Universal Robots PolyScope program: Floor Corner Extended.urp

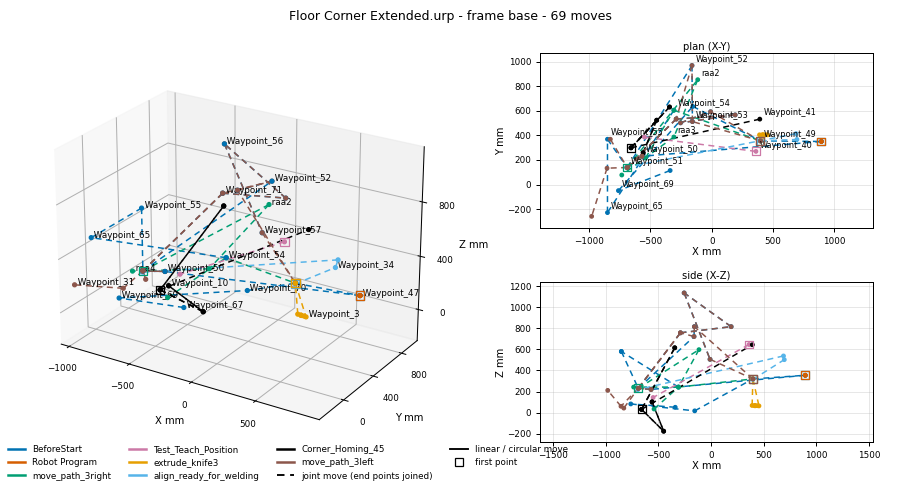
[picture p0: tool path of Floor Corner Extended.urp in frame base, 69 of 124 moves have a stored position in this frame; points joined in program order, loops and branches not executed]
Program Floor Corner Extended (installation=default directory=/programs/UPF createdIn=5.14.5 lastSavedIn=5.14.5 robotSerialNumber=20236801216)
Calibrated DH parameters: a=[-0.000021, -0.748897, -0.28186, -0.00004, -0.000055, 0]; d=[0.236225, -424.082933, -1564.66872, 1988.95162, 0.159094, 0.153873]; alpha=[1.570844, 0.001002, 0.000337, 1.571488, -1.569996, 0]; deltaTheta=[0, -0.516316, 5.626292, 1.173211, 0.000001, 0]
InitVariablesNode variables(variable(name=freedrive_m_var, expression=False))
BeforeStart
  Folder Safe Home Folder
    'if robot is not at home, send it back to home safely'
    'make sure the tcp is welder'
    Set NoAction tcp=pretend_welder
    sp := get_actual_tcp_pose()
    MoveL speed 250 mm/s, acceleration 1200 mm/s^2 (useActiveTCP=true) feature=Base
      Waypoint Variable (Variable): variable=sp
      'if first move is to a variable, skip automove'
    'turn off welder'
    URCap WireTank Serial (WireTank Serial, WireTank, LLC) dataModel(NODE_TITLE=Serial Bridge uR0, Command=[252,82,48], byte_array=true, OUTPUT_ENTRY=Static, QUERY=false, Variable(key=OUTPUT_VARIABLE, variable(name=HwResp)))
    Set DigitalOutput pin=digital_out[0]; digitalValue=0
    jp := get_actual_joint_positions()
    If sp[0]>0.600
      'if x > 600 then above then home'
      MoveJ speed 60 deg/s, acceleration 80 deg/s^2 (useActiveTCP=true) feature=Base
        Waypoint Waypoint_47: TCP in base x=894.111 y=351.078 z=354.441 mm, rx=2.3264 ry=2.0525 rz=0.0574 rad; joints [-187.182, -67.293, 94.726, 57.522, -0.141, -88.018] deg; TCP offset x=-5.49 y=-328 z=106.39 mm, rx=1.2092 ry=-1.2092 rz=1.2092 rad
      SafeHome (positionOptionType=SPEED_AND_ACCELERATION speed=1.047198 acceleration=1.396263 nextMotionTime=2)
    Else 
      Popup Message (haltProgram=false message=retreating to home inputType=Text)
      'for rules 2-8, finish with oldhome then above then home'
      If -1.74<jp[4] and jp[4]<1.05 and -1.74<jp[3] and jp[3]<1.74
        'if oldhome, test teach, then go straight to oldhome'
      ElseIf sp[0]<-.5 and jp[3]>3.14 and -2.62<jp[4] and jp[4]<-0.87
        'if left side weld approach, left weld approach in reverse'
        MoveJ speed 60 deg/s, acceleration 80 deg/s^2 (useActiveTCP=true) feature=Base
          Waypoint Waypoint_50: TCP in base x=-568.711 y=230.602 z=220.209 mm, rx=-1.5191 ry=-0.5351 rz=0.574 rad; joints [-1.233, -73.308, 139.365, 291.685, -131.758, 87.871] deg
          Waypoint Waypoint_51: TCP in base x=-689.65 y=139.001 z=230.693 mm, rx=-0.852 ry=-1.646 rz=1.646 rad; joints [-65.631, -88.39, 163.033, 285.278, -280.919, 90.062] deg
          Waypoint Waypoint_52: TCP in base x=-160.992 y=970.528 z=722.037 mm, rx=-0.555 ry=0.1065 rz=0.3285 rad; joints [-74.362, -75.728, 129.393, 212.138, -169.184, 55.164] deg
          Waypoint Waypoint_53: TCP in base x=-157.624 y=513.351 z=815.67 mm, rx=-0.6727 ry=-1.8523 rz=-0.0554 rad; joints [-158.576, -104.315, 132.512, 57.998, -61.68, -46.426] deg
      ElseIf sp[0]<0 and 0<jp[3] and jp[3]<1.74 and 0.87<jp[4] and jp[4]<2.62
        'if right side around, move back then wapoint 24 then oldhome'
        If sp[0]<-1.0
          xback := p[-1.0,sp[1],sp[2],sp[3],sp[4],sp[5]]
          MoveJ speed 60 deg/s, acceleration 80 deg/s^2 (useActiveTCP=true) feature=Base
            Waypoint Variable (Variable): variable=xback
        MoveJ speed 60 deg/s, acceleration 80 deg/s^2 (useActiveTCP=true) feature=Base
          Waypoint Waypoint_54: TCP in base x=-308.528 y=606.081 z=242.371 mm, rx=-2.1337 ry=0.3494 rz=2.131 rad; joints [-112.4, -74.451, 126.505, 42.726, 91.418, 81.282] deg
      ElseIf jp[3]>2.62 and jp[4]<-3.84
        'if left side second half, then left weld ending sequence'
        If jp[5]<0.35
          MoveJ speed 60 deg/s, acceleration 80 deg/s^2 (useActiveTCP=true) feature=Base
            Waypoint Waypoint_65: TCP in base x=-850.3 y=-229.061 z=580.194 mm, rx=-0.0667 ry=-1.5664 rz=-0.0455 rad; joints [6.605, -69.14, 152.414, 186.359, -269.256, -10.612] deg
        MoveJ speed 60 deg/s, acceleration 80 deg/s^2 (useActiveTCP=true) feature=Base
          SuppressedNode
            Waypoint Waypoint_61: TCP in base x=-1224.453 y=315.135 z=45.036 mm, rx=0.4556 ry=-1.5209 rz=0.4778 rad; joints [-38.105, -18.537, 102.715, 186.465, -269.531, 72.317] deg
          SuppressedNode
            Waypoint Waypoint_62: TCP in base x=-1246.058 y=121.907 z=25.888 mm, rx=-0.7807 ry=-1.4195 rz=-0.7637 rad; joints [-2.239, -16.844, 100.196, 185.863, -269.635, -54.527] deg
          SuppressedNode
            Waypoint Waypoint_63: TCP in base x=-850.3 y=142.696 z=580.194 mm, rx=-0.0667 ry=-1.5664 rz=-0.0455 rad; joints [-33.715, -70.118, 156.539, 183.763, -269.222, 29.711] deg
          SuppressedNode
            Waypoint Waypoint_64: TCP in base x=-850.307 y=-229.065 z=580.197 mm, rx=-0.0667 ry=-1.5664 rz=-0.0455 rad; joints [6.605, -69.141, 152.414, 186.36, -269.255, -10.612] deg
          'above is testing, below is real'
          Waypoint Waypoint_55: TCP in base x=-850.296 y=369.354 z=580.191 mm, rx=-0.0667 ry=-1.5664 rz=-0.0455 rad; joints [-51.358, -68.674, 149.321, 189.759, -269.326, 47.358] deg
          SuppressedNode
            Waypoint Waypoint_60: TCP in base x=-826.865 y=369.366 z=43.112 mm, rx=0.575 ry=-1.4922 rz=0.5971 rad; joints [-59.177, -17.074, 121.534, 166.294, -269.929, 102.173] deg
          Waypoint Waypoint_59: motionParameters(nextMotionTime=2); TCP in base x=-689.651 y=138.973 z=230.7 mm, rx=-0.852 ry=-1.646 rz=1.646 rad; joints [-65.63, -88.392, 163.034, 285.278, -280.919, 90.062] deg
          Waypoint Waypoint_71: TCP in base x=-289.685 y=534.258 z=757.199 mm, rx=-0.2952 ry=-0.653 rz=0.3894 rad; joints [-79.881, -94.829, 156.624, 238.16, -217.621, 99.184] deg
          Waypoint Waypoint_58: TCP in base x=191.12 y=567.518 z=815.513 mm, rx=-0.1358 ry=0.3961 rz=0.2088 rad; joints [-94.611, -101.484, 149.999, 189.458, -152.19, 49.064] deg
          Waypoint Waypoint_56: TCP in base x=-254.568 y=502.959 z=1135.401 mm, rx=-0.2619 ry=-0.7497 rz=1.3491 rad; joints [-116.567, -108.934, 141.5, 126.12, -66.905, -29.189] deg
          Waypoint Waypoint_57: TCP in base x=-9.221 y=593.713 z=505.809 mm, rx=-1.4244 ry=-2.3441 rz=-0.5276 rad; joints [-167.352, -114.202, 136.688, 39.052, -32.592, -65.93] deg
      ElseIf jp[3]<-2.09
        'bottom homing'
        MoveJ speed 60 deg/s, acceleration 80 deg/s^2 (useActiveTCP=true) feature=Base
          SuppressedNode
            Waypoint Waypoint_66: TCP in base x=-1189.333 y=-102.843 z=-176.058 mm, rx=1.1963 ry=-1.1853 rz=1.2301 rad; joints [-19.887, -1.876, 78.341, -165.92, 91.498, 110.543] deg
          ''
          If sp[0]<-0.95
            xback := p[-0.95,sp[1],sp[2],sp[3],sp[4],sp[5]]
            MoveL speed 250 mm/s, acceleration 1200 mm/s^2 (useActiveTCP=true) feature=Base
              Waypoint Variable (Variable): variable=xback
          Waypoint Waypoint_67: TCP in base x=-339.169 y=114.271 z=51.007 mm, rx=-0.4342 ry=1.8727 rz=-1.8852 rad; joints [-80.817, -56.025, 141.954, -98.756, -22.671, 103.625] deg
      ElseIf jp[3]<0 and jp[4]<-3.14
        'if left side homing, special unspin'
        MoveJ speed 60 deg/s, acceleration 80 deg/s^2 (useActiveTCP=true) feature=Base
          SuppressedNode
            Waypoint Waypoint_68: TCP in base x=-1436.144 y=-207.487 z=20.65 mm, rx=-1.0168 ry=-1.7024 rz=1.6295 rad; joints [2.271, -43.137, 96.498, -42.2, -211.884, 93.908] deg
          ''
          Waypoint Waypoint_69: TCP in base x=-760.827 y=-49.763 z=82.65 mm, rx=-1.0262 ry=-1.6127 rz=1.5471 rad; joints [-12.694, -64.084, 157.914, -89.201, -220.703, 89.352] deg
          Waypoint Waypoint_70: TCP in base x=-154.415 y=636.923 z=16.979 mm, rx=-0.3028 ry=1.487 rz=0.1222 rad; joints [-64.641, -61.184, 139.176, -160.395, -91.873, 99.702] deg
      ElseIf (sp[4]<-3 or sp[4]>3) and -0.02<sp[5] and sp[5]<0.02
        'go straight to home'
      ElseIf 2>1
        'if none of the other options, then error continuously'
        Loop While (checkContinuously=false) expression=2>1
          Popup Message (haltProgram=false message=Unknown Position. Find Calvin for Assistance inputType=Text)
      'insert logic for how to get back to oldhome'
      'finish with oldhome then above then home'
      MoveJ speed 60 deg/s, acceleration 80 deg/s^2 (useActiveTCP=true) feature=Base
        Waypoint Waypoint_49: motionParameters(jointSpeed=1.047198 jointAcceleration=1.396263 cartesianSpeed=0.25 cartesianAcceleration=1.2); TCP in base x=397.354 y=356.263 z=319.809 mm, rx=2.3163 ry=2.0576 rz=0.0741 rad; joints [-198.126, -117.851, 133.304, -13.008, -11.424, -6.036] deg
        Waypoint Waypoint_48: TCP in base x=894.09 y=351.09 z=354.453 mm, rx=2.3264 ry=2.0525 rz=0.0573 rad; joints [-187.181, -67.294, 94.727, 57.523, -0.141, -88.018] deg
      SafeHome (positionOptionType=SPEED_AND_ACCELERATION speed=1.047198 acceleration=1.396263 nextMotionTime=2)
Robot Program (runOnlyOnce=true)
  'start of main program'
  Set NoAction tcp=pretend_welder
  SafeHome (positionOptionType=SPEED_AND_ACCELERATION speed=1.047198 acceleration=1.396263 nextMotionTime=2)
  Script file /programs/analyze_touchpoints.script
    | # this file creates the function for analyzing touchpoints
    | # define pi
    | pi = 3.1415926535
    | 
    | # this is the main entry point for calculations.
    | # it takes in the 5 points, analyzes the shape of the box, and then calculates path points and returns them
    | # specifically for Down, Over, then Around (DOtA)
    | # specifically for right-sided boxes (vertical weld on right side of edge)
    | def main_calculate_right(p11, p12, p21, p22, p3, p13, p23, chamferover):
    |     struct1 = analyze_touchpoints_only(p11, p12, p21, p22, p3)
    |     list1 = analyze_vertical_touchpoints(p11, p12, p13, p21, p22, p23, p3)
    |     struct2 = calculate_DOtA_points_right(struct1, list1, chamferover)
    |     validity = check_validity_right(struct1, struct2)
    |     return struct2
    | end
    | 
    | # this is the main entry point for calculations.
    | # it takes in the 5 points, analyzes the shape of the box, and then calculates path points and returns them
    | # specifically for Down, Over, then Around (DOtA)
    | # specifically for left-sided boxes (vertical weld on left side of edge)
    | def main_calculate_left(p11, p12, p21, p22, p3, p13, p23, chamferover):
    |     struct1 = analyze_touchpoints_only(p11, p12, p21, p22, p3)
    |     list1 = analyze_vertical_touchpoints(p11, p12, p13, p21, p22, p23, p3)
    |     struct2 = calculate_DOtA_points_left(struct1, list1, chamferover)
    |     validity = check_validity_left(struct1, struct2)
    |     return struct2
    | end
    | 
    | # this is the main entry point for calculations, for Floor Corner Extended.
    | # it takes in the 7 touchpoints, analyzes the shape of the box.
    | # takes in the user defined point for the top of the weld (tcp_pose_top) and then calculates path points
    | # loopingly tries to calculate the extension along the sidewall that fulfills get_inverse_kin_has_solution() and provides the farthest extension possible
    | # returns the pathpoints
    | # specifically for Down, Over, then Around (DOtA)
    | # specifically for right-sided boxes (vertical weld on right side of edge)
    | def main_calculate_right_extended(p11, p12, p21, p22, p3, p13, p23, chamferover, tcp_pose_top):
    |     struct1 = analyze_touchpoints_only(p11, p12, p21, p22, p3)
    |     list1 = analyze_vertical_touchpoints(p11, p12, p13, p21, p22, p23, p3)
    |     struct2 = calculate_DOtA_points_right_extended(struct1, list1, chamferover, tcp_pose_top)
    |     validity = check_validity_right(struct1, struct2)
    |     return struct2
    | end
    | 
    | # this is the main entry point for calculations, for Floor Corner Extended.
    | # it takes in the 7 touchpoints, analyzes the shape of the box.
    | # takes in the user defined point for the top of the weld (tcp_pose_top) and then calculates path points
    | # loopingly tries to calculate the extension along the sidewall that fulfills get_inverse_kin_has_solution() and provides the farthest extension possible
    | # returns the pathpoints
    | # specifically for Down, Over, then Around (DOtA)
    | # specifically for left-sided boxes (vertical weld on left side of edge)
    | def main_calculate_left_extended(p11, p12, p21, p22, p3, p13, p23, chamferover, tcp_pose_top):
    |     struct1 = analyze_touchpoints_only(p11, p12, p21, p22, p3)
    |     list1 = analyze_vertical_touchpoints(p11, p12, p13, p21, p22, p23, p3)
    |     struct2 = calculate_DOtA_points_left_extended(struct1, list1, chamferover, tcp_pose_top)
    |     validity = check_validity_left(struct1, struct2)
    |     return struct2
    | end
    | 
    | # it takes 5 arguments as points
    | # it returns a struct containing: (pointintersect, pointapproach1, pointapproach2, point1, point2, point3, point4, point5, pointreturn1, heading1, heading2, heading3, path2r1, path2r2, path2l1, path2l2)
    | # specifically for Around then Up (AtU)
    | def analyze_touchpoints(p11, p12, p21, p22, p3):
    |   # FIND THE INTERSECTION
    |   # comment get the z
    |   zcoord=p3[2]
    | 
    |   # get the raw points from the first line
    |   l1p1x=p11[0]
    |   l1p1y=p11[1]
    |   l1p2x=p12[0]
    |   l1p2y=p12[1]
    | 
    |   # equate the first line in 2d space
    |   ml1 = (l1p2y-l1p1y) / (l1p2x-l1p1x)
    | 
    |   # b = y - mx
    |   bl1 = l1p1y - ml1 * l1p1x
    | 
    |   # get the raw points from the second line
    |   l2p1x=p21[0]
    |   l2p1y=p21[1]
    |   l2p2x=p22[0]
    |   l2p2y=p22[1]
    | 
    |   # equate the second line in 2d space
    |   ml2 = (l2p2y-l2p1y) / (l2p2x-l2p1x)
    | 
    |   # b = y - mx
    |   bl2 = l2p1y - ml2 * l2p1x
    | 
    | 
    |   # find the intersection of the two lines
    |   # m1x+b1 = m2x+b2
    |   # m1x - m2x = b2 - b1
    |   # x = (b2-b1) / (m1-m2)
    |   xintersect = (bl2-bl1) / (ml1-ml2)
    |   yintersect = ml1 * xintersect + bl1
    | 
    |   #FIND THE VECTORS
    |   #define a vector from the intersection to the second point on the first line
    |   l1delxfull = l1p2x - xintersect
    |   l1delyfull = l1p2y - yintersect
    | 
    |   l1delmag = sqrt(l1delxfull*l1delxfull + l1delyfull*l1delyfull)
    | 
    |   l1delxunit = l1delxfull / l1delmag
    |   l1delyunit = l1delyfull / l1delmag
    | 
    |   #define a vector from the intersection to the second point on the second line
    |   l2delxfull = l2p2x - xintersect
    |   l2delyfull = l2p2y - yintersect
    | 
    |   l2delmag = sqrt(l2delxfull*l2delxfull + l2delyfull*l2delyfull)
    | 
    |   l2delxunit = l2delxfull / l2delmag
    |   l2delyunit = l2delyfull / l2delmag
    | 
    |   # FIND THE FOUR POINTS ON THE LINES
    |   # find locations 8 inches away from  intersect point
    |   # CONST
    |   welddistance = 8
    |   roundoverdistance = 0.05
    |   zup = .375
    |   # inches
    |   wd = welddistance * 25.4 / 1000
    |   rod = roundoverdistance * 25.4 / 1000
    |   zup = zup * 25.4 / 1000
    | 
    |   # now we have the unit vector. extend the weld distance from the intersection
    |   x = xintersect + l1delxunit * wd
    |   y = yintersect + l1delyunit * wd
    |   z = zcoord + zup
    | 
    |   point1 = p[x,y,z,1.570796,0,0] # dummy orientation for now
    | 
    |   x = xintersect + l1delxunit * rod
    |   y = yintersect + l1delyunit * rod
    | 
    |   point2 = p[x,y,z,1.570796,0,0]
    | 
    |   # now we have the unit vector. extend the weld distance from the intersection
    |   x = xintersect + l2delxunit * wd
    |   y = yintersect + l2delyunit * wd
    | 
    |   point5 = p[x,y,z,0,-1.570796,0]
    | 
    |   x = xintersect + l2delxunit * rod
    |   y = yintersect + l2delyunit * rod
    | 
    |   point4 = p[x,y,z,0,-1.570796,0]
    | 
    |   #DEFINE APPROACH POINTS
    |   pointintersect = p[xintersect,yintersect,zcoord,0,0,0]
    |   pointapproach1 = p[xintersect+0.1,yintersect+0.1,z,1.570796,0,0]
    |   pointapproach2 = p[point1[0], point1[1]+0.1, point1[2], point1[3], point1[4], point1[5]]
    |   pointreturn1 = p[point5[0]+0.1, point5[1], point5[2], point5[3], point5[4], point5[5]]
    | 
    |   #FIND HEADINGS
    |   #for each heading, find the angle of the line with respect to the pos x axis. then add/subtract 90 degrees because you want to be perpendicular to that
    |   headingvector1 = convert_uv_to_heading(l1delxunit, l1delyunit)
    |   headingvector2 = convert_uv_to_heading(l2delxunit, l2delyunit)
    |   # find halfway heading
    |   heading2 = (headingvector1 + headingvector2)/2
    |   # find headings that the robot should face while traveling, perpendicular to the vectors of the sides of the box
    |   heading1 = headingvector1 + pi/2
    |   heading3 = headingvector2 - pi/2
    | 
    |   #FIND POINT 3
    |   #see if we have to / can find point 3
    |   findpoint3 = True
    |   if roundoverdistance == 0:
    |     findpoint3 = False
    |   end
    |   if findpoint3:
    |     # i need to find the point3 such that the arc from p2 to p3 to p4 is tangent to p1-p2 and p4-p5. making this a smooth path will be good
    |     # the direction of movement is from pointintersect in the direction of heading2
    |     # how much movement though? this will depend on whether it is actually a 90 degree angle or not.
    |     # first, find the perpendicular lines through points 2 and 4
    |     perp2 = find_perpendicular_line(ml1, point2[0], point2[1])
    |     perp4 = find_perpendicular_line(ml2, point4[0], point4[1])
    |     # next, find the intersection of those two lines
    |     perpintersect = find_intersection(perp2[0], perp2[1], perp4[0], perp4[1])
    |     radiusofcircle = distance_between(perpintersect[0], perpintersect[1], 0, point2[0], point2[1], 0)
    |     # find a vector the direction of heading2
    |     uvx = cos(heading2)
    |     uvy = sin(heading2)
    |     # compute point3. pass in negative radius because the direction is into the tank but we want to move from the intersection out to the rounded edge
    |     point3coords = add_vectordistance_to_point(perpintersect[0], perpintersect[1], z, uvx, uvy, 0, -1 * radiusofcircle)
    |     point3 = p[point3coords[0], point3coords[1], point3coords[2], 0, 0, 0]
    |   end
    | 
    |   #APPLY ACTUAL RXRYRZ TO POINTS
    |   # convert the headings to rxryrz and insert those values into the relevant points
    |   rxryrz = convert_heading_to_axang(heading1)
    |   rx = rxryrz[0]
    |   ry = rxryrz[1]
    |   rz = rxryrz[2]
    |   pointapproach1 = p[pointapproach1[0], pointapproach1[1], pointapproach1[2], rx, ry, rz]
    |   pointapproach2 = p[pointapproach2[0], pointapproach2[1], pointapproach2[2], rx, ry, rz]
    |   point1 = p[point1[0], point1[1], point1[2], rx, ry, rz]
    |   point2 = p[point2[0], point2[1], point2[2], rx, ry, rz]
    |   rxryrz = convert_heading_to_axang(heading2)
    |   rx = rxryrz[0]
    |   ry = rxryrz[1]
    |   rz = rxryrz[2]
    |   if findpoint3:
    |     point3 = p[point3[0], point3[1], point3[2], rx, ry, rz]
    |   else:
    |     point3 = point2
    |   end
    |   rxryrz = convert_heading_to_axang(heading3)
    |   rx = rxryrz[0]
    |   ry = rxryrz[1]
    |   rz = rxryrz[2]
    |   point4 = p[point4[0], point4[1], point4[2], rx, ry, rz]
    |   point5 = p[point5[0], point5[1], point5[2], rx, ry, rz]
    |   pointreturn1 = p[pointreturn1[0], pointreturn1[1], pointreturn1[2], rx, ry, rz]
    | 
    |   #find path2 (the part that goes up)
    |   four_vertical_points = find_vertical_points(pointintersect, l1delxunit, l1delyunit, l2delxunit, l2delyunit, zup, wd, heading1, heading3)
    |   path2r1 = four_vertical_points[0]
    |   path2r2 = four_vertical_points[1]
    |   path2l1 = four_vertical_points[2]
    |   path2l2 = four_vertical_points[3]
    | 
    |   #RETURN STRUCT
    |   ret = struct(pointintersect=pointintersect, pointapproach1=pointapproach1, pointapproach2=pointapproach2, point1=point1, point2=point2, point3=point3, point4=point4, point5=point5, pointreturn1=pointreturn1, heading1=heading1, heading2=heading2, heading3=heading3, path2r1=path2r1, path2r2=path2r2, path2l1=path2l1, path2l2=path2l2)
    |   return ret
    | end
    | 
    | # it takes 5 arguments as points
    | # it returns a struct containing: (pointintersect, heading1, heading2, heading3, l1delxunit, l1delyunit, l2delxunit, l2delyunit)
    | def analyze_touchpoints_only(p11, p12, p21, p22, p3):
    |   # FIND THE INTERSECTION
    |   # comment get the z
    |   zcoord=p3[2]
    | 
    |   # get the raw points from the first line
    |   l1p1x=p11[0]
    |   l1p1y=p11[1]
    |   l1p2x=p12[0]
    |   l1p2y=p12[1]
    | 
    |   # equate the first line in 2d space
    |   ml1 = (l1p2y-l1p1y) / (l1p2x-l1p1x)
    | 
    |   # b = y - mx
    |   bl1 = l1p1y - ml1 * l1p1x
    | 
    |   # get the raw points from the second line
    |   l2p1x=p21[0]
    |   l2p1y=p21[1]
    |   l2p2x=p22[0]
    |   l2p2y=p22[1]
    | 
    |   # equate the second line in 2d space
    |   ml2 = (l2p2y-l2p1y) / (l2p2x-l2p1x)
    | 
    |   # b = y - mx
    |   bl2 = l2p1y - ml2 * l2p1x
    | 
    | 
    |   # find the intersection of the two lines
    |   # m1x+b1 = m2x+b2
    |   # m1x - m2x = b2 - b1
    |   # x = (b2-b1) / (m1-m2)
    |   xintersect = (bl2-bl1) / (ml1-ml2)
    |   yintersect = ml1 * xintersect + bl1
    | 
    |   pointintersect = p[xintersect,yintersect,zcoord,0,0,0]
    | 
    |   #FIND THE VECTORS
    |   #define a vector from the intersection to the second point on the first line
    |   l1delxfull = l1p2x - xintersect
    |   l1delyfull = l1p2y - yintersect
    | 
    |   l1delmag = sqrt(l1delxfull*l1delxfull + l1delyfull*l1delyfull)
    | 
    |   l1delxunit = l1delxfull / l1delmag
    |   l1delyunit = l1delyfull / l1delmag
    | 
    |   #define a vector from the intersection to the second point on the second line
    |   l2delxfull = l2p2x - xintersect
    |   l2delyfull = l2p2y - yintersect
    | 
    |   l2delmag = sqrt(l2delxfull*l2delxfull + l2delyfull*l2delyfull)
    | 
    |   l2delxunit = l2delxfull / l2delmag
    |   l2delyunit = l2delyfull / l2delmag
    | 
    |   #FIND HEADINGS
    |   #for each heading, find the angle of the line with respect to the pos x axis. then add/subtract 90 degrees because you want to be perpendicular to that
    |   headingvector1 = convert_uv_to_heading(l1delxunit, l1delyunit)
    |   headingvector2 = convert_uv_to_heading(l2delxunit, l2delyunit)
    |   # find halfway heading
    |   heading2 = (headingvector1 + headingvector2)/2
    |   # find headings that the robot should face while traveling, perpendicular to the vectors of the sides of the box
    |   heading1 = headingvector1 + pi/2
    |   heading3 = headingvector2 - pi/2
    | 
    |   #RETURN STRUCT
    |   ret = struct(pointintersect=pointintersect, heading1=heading1, heading2=heading2, heading3=heading3, l1delxunit=l1delxunit, l1delyunit=l1delyunit, l2delxunit=l2delxunit, l2delyunit=l2delyunit)
    |   return ret
    | end
    | 
    | # given a struct from analyze_touchpoints_only(), calculate the points
    | # for right, for non-extended
    | def calculate_DOtA_points_right(struct1, listleans, chamferover):
    |     # get the stuff from the struct
    |     pointintersect = struct1[0]
    |     heading1 = struct1[1]
    |     heading2 = struct1[2]
    |     heading3 = struct1[3]
    |     l1delxunit = struct1[4]
    |     l1delyunit = struct1[5]
    |     l2delxunit = struct1[6]
    |     l2delyunit = struct1[7]
    | 
    |     # FIND THE POINTS ON THE LINES OF THE FIRST TURN PATH
    |     # find locations 8 inches away from  intersect point
    |     # CONST
    |     welddistance1 = 8 # vertical weld distance
    |     welddistance2 = 6 # first path second leg
    |     welddistance3 = 8 # second path second leg
    |     zup = .375
    |     # inches
    |     wd1 = welddistance1 * 25.4 / 1000
    |     wd2 = welddistance2 * 25.4 / 1000
    |     wd3 = welddistance3 * 25.4 / 1000
    |     zup = zup * 25.4 / 1000
    |     chamferovermm =  chamferover * 25.4 / 1000
    | 
    |     x = pointintersect[0] + l1delxunit * chamferovermm
    |     y = pointintersect[1] + l1delyunit * chamferovermm
    |     z = pointintersect[2] + zup
    | 
    |     #apply actual rxryrz to points
    |     # convert the headings to rxryrz and insert those values into the relevant points
    |     rxryrz = convert_heading_to_axang_preheatdown(heading1)
    |     rx = rxryrz[0]
    |     ry = rxryrz[1]
    |     rz = rxryrz[2]
    | 
    |     point1 = p[x + wd1*listleans[0], y + wd1*listleans[1], z + wd1, rx, ry, rz] # add in the listleans factor to follow the face of the box as we move up
    |     point2 = p[x, y, z, rx, ry, rz]
    | 
    |     # convert the headings to rxryrz and insert those values into the relevant points
    |     rxryrz = convert_heading_to_axang_ccw(heading1)
    |     rx = rxryrz[0]
    |     ry = rxryrz[1]
    |     rz = rxryrz[2]
    | 
    |     point4 = p[x, y, z, rx, ry, rz]
    |     x = x + l1delxunit * wd2
    |     y = y + l1delyunit * wd2
    |     point5 = p[x, y, z, rx, ry, rz]
    | 
    |     # FIND THE POINTS ON THE LINES OF THE SECOND AROUND PATH
    |     roundoverdistance = 0.05
    |     rod = roundoverdistance * 25.4 / 1000
    | 
    |     # now we have the unit vector. extend the weld distance from the intersection
    |     x = pointintersect[0] + l1delxunit * chamferovermm
    |     y = pointintersect[1] + l1delyunit * chamferovermm
    |     # convert the headings to rxryrz and insert those values into the relevant points
    |     rxryrz = convert_heading_to_axang(heading1)
    |     rx = rxryrz[0]
    |     ry = rxryrz[1]
    |     rz = rxryrz[2]
    |     point_1 = p[x, y, z, rx, ry, rz]
    | 
    |     x = pointintersect[0] + l1delxunit * rod
    |     y = pointintersect[1] + l1delyunit * rod
    |     point_2 = p[x, y, z, rx, ry, rz]
    | 
    |     # now we have the unit vector. extend the weld distance from the intersection
    |     x = pointintersect[0] + l2delxunit * wd3
    |     y = pointintersect[1] + l2delyunit * wd3
    |     # convert the headings to rxryrz and insert those values into the relevant points
    |     rxryrz = convert_heading_to_axang(heading3)
    |     rx = rxryrz[0]
    |     ry = rxryrz[1]
    |     rz = rxryrz[2]
    |     point_5 = p[x, y, z, rx, ry, rz]
    | 
    |     x = pointintersect[0] + l2delxunit * rod
    |     y = pointintersect[1] + l2delyunit * rod
    |     point_4 = p[x, y, z, rx, ry, rz]
    | 
    |     #FIND POINT 3
    |     # by calling analyze_touchpoints()
    |     atret = analyze_touchpoints(point_2, point_1, point_4, point_5, pointintersect)
    |     point_3 = atret[5]
    | 
    | 
    |     struct2 = struct(point1=point1, point2=point2, point4=point4, point5=point5, point_1=point_1, point_2=point_2, point_3=point_3, point_4=point_4, point_5=point_5)
    |     return struct2
    | end
    | 
    | # given a struct from analyze_touchpoints_only(), calculate the points
    | # for left, for non-extended
    | def calculate_DOtA_points_left(struct1, listleans, chamferover):
    |     # get the stuff from the struct
    |     pointintersect = struct1[0]
    |     heading1 = struct1[1]
    |     heading2 = struct1[2]
    |     heading3 = struct1[3]
    |     l1delxunit = struct1[4]
    |     l1delyunit = struct1[5]
    |     l2delxunit = struct1[6]
    |     l2delyunit = struct1[7]
    | 
    |     # FIND THE POINTS ON THE LINES OF THE FIRST TURN PATH
    |     # find locations 8 inches away from  intersect point
    |     # CONST
    |     welddistance1 = 8 # vertical weld distance
    |     welddistance2 = 6 # first path second leg
    |     welddistance3 = 8 # second path second leg
    |     zup = .375
    |     # inches
    |     wd1 = welddistance1 * 25.4 / 1000
    |     wd2 = welddistance2 * 25.4 / 1000
    |     wd3 = welddistance3 * 25.4 / 1000
    |     zup = zup * 25.4 / 1000
    |     chamferovermm =  chamferover * 25.4 / 1000
    | 
    |     x = pointintersect[0] + l2delxunit * chamferovermm
    |     y = pointintersect[1] + l2delyunit * chamferovermm
    |     z = pointintersect[2] + zup
    | 
    |     #apply actual rxryrz to points
    |     # convert the headings to rxryrz and insert those values into the relevant points
    |     rxryrz = convert_heading_to_axang_preheatdown(heading3)
    |     rx = rxryrz[0]
    |     ry = rxryrz[1]
    |     rz = rxryrz[2]
    | 
    |     point1 = p[x + wd1*listleans[0], y + wd1*listleans[1], z + wd1, rx, ry, rz]
    |     point2 = p[x, y, z, rx, ry, rz]
    | 
    |     # convert the headings to rxryrz and insert those values into the relevant points
    |     rxryrz = convert_heading_to_axang(heading3)
    |     rx = rxryrz[0]
    |     ry = rxryrz[1]
    |     rz = rxryrz[2]
    | 
    |     point4 = p[x, y, z, rx, ry, rz]
    |     x = x + l2delxunit * wd2
    |     y = y + l2delyunit * wd2
    |     point5 = p[x, y, z, rx, ry, rz]
    | 
    |     # FIND THE POINTS ON THE LINES OF THE SECOND AROUND PATH
    |     roundoverdistance = 0.05
    |     rod = roundoverdistance * 25.4 / 1000
    | 
    |     # now we have the unit vector. extend the weld distance from the intersection
    |     x = pointintersect[0] + l2delxunit * chamferovermm
    |     y = pointintersect[1] + l2delyunit * chamferovermm
    |     # convert the headings to rxryrz and insert those values into the relevant points
    |     rxryrz = convert_heading_to_axang_ccw(heading3)
    |     rx = rxryrz[0]
    |     ry = rxryrz[1]
    |     rz = rxryrz[2]
    |     point_1 = p[x, y, z, rx, ry, rz]
    | 
    |     x = pointintersect[0] + l2delxunit * rod
    |     y = pointintersect[1] + l2delyunit * rod
    |     point_2 = p[x, y, z, rx, ry, rz]
    | 
    |     # now we have the unit vector. extend the weld distance from the intersection
    |     x = pointintersect[0] + l1delxunit * wd3
    |     y = pointintersect[1] + l1delyunit * wd3
    |     # convert the headings to rxryrz and insert those values into the relevant points
    |     rxryrz = convert_heading_to_axang_ccw(heading1)
    |     rx = rxryrz[0]
    |     ry = rxryrz[1]
    |     rz = rxryrz[2]
    |     point_5 = p[x, y, z, rx, ry, rz]
    | 
    |     x = pointintersect[0] + l1delxunit * rod
    |     y = pointintersect[1] + l1delyunit * rod
    |     point_4 = p[x, y, z, rx, ry, rz]
    | 
    |     #FIND POINT 3
    |     # by calling analyze_touchpoints()
    |     atret = analyze_touchpoints(point_2, point_1, point_4, point_5, pointintersect)
    |     point_3 = atret[5]
    |     #point 3 will not have the correct rxryrz though because now the gun needs to be face up.
    |     rxryrz = convert_heading_to_axang_ccw(heading2)
    |     rx = rxryrz[0]
    |     ry = rxryrz[1]
    |     rz = rxryrz[2]
    |     point_3 = p[point_3[0], point_3[1], point_3[2], rx, ry, rz]
    | 
    |     struct2 = struct(point1=point1, point2=point2, point4=point4, point5=point5, point_1=point_1, point_2=point_2, point_3=point_3, point_4=point_4, point_5=point_5)
    |     return struct2
    | end
    | 
    | # given a struct from analyze_touchpoints_only(), calculate the points
    | # for right, for extended
    | def calculate_DOtA_points_right_extended(struct1, listleans, chamferover, tcp_pose_top):
    |     # get the stuff from the struct
    |     pointintersect = struct1[0]
    |     heading1 = struct1[1]
    |     heading2 = struct1[2]
    |     heading3 = struct1[3]
    |     l1delxunit = struct1[4]
    |     l1delyunit = struct1[5]
    |     l2delxunit = struct1[6]
    |     l2delyunit = struct1[7]
    | 
    |     # FIND THE POINTS ON THE LINES OF THE FIRST TURN PATH
    |     # find locations 8 inches away from  intersect point
    |     # CONST
    |     # welddistance1 = 8 # vertical weld distance
    |     welddistance2 = 6 # first path second leg
    |     welddistance3 = 8 # second path second leg
    |     zup = .375
    |     # inches
    |     # wd1 = welddistance1 * 25.4 / 1000
    |     wd2 = welddistance2 * 25.4 / 1000
    |     wd3 = welddistance3 * 25.4 / 1000
    |     zup = zup * 25.4 / 1000
    |     chamferovermm =  chamferover * 25.4 / 1000
    | 
    |     # weld distance is the distance that it will weld. this will make it start at the z height that the user specified
    |     wd1 = tcp_pose_top[2] - pointintersect[2] - zup
    | 
    |     x = pointintersect[0] + l1delxunit * chamferovermm
    |     y = pointintersect[1] + l1delyunit * chamferovermm
    |     z = pointintersect[2] + zup
    | 
    |     #apply actual rxryrz to points
    |     # convert the headings to rxryrz and insert those values into the relevant points
    |     rxryrz = convert_heading_to_axang_preheatdown(heading1)
    |     rx = rxryrz[0]
    |     ry = rxryrz[1]
    |     rz = rxryrz[2]
    | 
    |     point1 = p[x + wd1*listleans[0], y + wd1*listleans[1], z + wd1, rx, ry, rz] # add in the listleans factor to follow the face of the box as we move up
    |     point2 = p[x, y, z, rx, ry, rz]
    | 
    |     # convert the headings to rxryrz and insert those values into the relevant points
    |     rxryrz = convert_heading_to_axang_ccw(heading1)
    |     rx = rxryrz[0]
    |     ry = rxryrz[1]
    |     rz = rxryrz[2]
    | 
    |     point4 = p[x, y, z, rx, ry, rz]
    |     x = x + l1delxunit * wd2
    |     y = y + l1delyunit * wd2
    |     point5 = p[x, y, z, rx, ry, rz]
    | 
    |     # FIND THE POINTS ON THE LINES OF THE SECOND AROUND PATH
    |     roundoverdistance = 0.05
    |     rod = roundoverdistance * 25.4 / 1000
    | 
    |     # now we have the unit vector. extend the weld distance from the intersection
    |     x = pointintersect[0] + l1delxunit * chamferovermm
    |     y = pointintersect[1] + l1delyunit * chamferovermm
    |     # convert the headings to rxryrz and insert those values into the relevant points
    |     rxryrz = convert_heading_to_axang(heading1)
    |     rx = rxryrz[0]
    |     ry = rxryrz[1]
    |     rz = rxryrz[2]
    |     point_1 = p[x, y, z, rx, ry, rz]
    | 
    |     x = pointintersect[0] + l1delxunit * rod
    |     y = pointintersect[1] + l1delyunit * rod
    |     point_2 = p[x, y, z, rx, ry, rz]
    | 
    |     # convert the headings to rxryrz and insert those values into the relevant points
    |     rxryrz = convert_heading_to_axang(heading3)
    |     rx = rxryrz[0]
    |     ry = rxryrz[1]
    |     rz = rxryrz[2]
    | 
    |     x = pointintersect[0] + l2delxunit * rod
    |     y = pointintersect[1] + l2delyunit * rod
    |     point_4 = p[x, y, z, rx, ry, rz]
    | 
    |     # now we have the unit vector. extend the weld distance from the intersection
    |     x = pointintersect[0] + l2delxunit * wd3
    |     y = pointintersect[1] + l2delyunit * wd3
    |     point_5 = p[x, y, z, rx, ry, rz]
    | 
    |     #FIND POINT 3
    |     # by calling analyze_touchpoints()
    |     atret = analyze_touchpoints(point_2, point_1, point_4, point_5, pointintersect)
    |     point_3 = atret[5]
    | 
    | 
    |     struct2 = struct(point1=point1, point2=point2, point4=point4, point5=point5, point_1=point_1, point_2=point_2, point_3=point_3, point_4=point_4, point_5=point_5)
    |     return struct2
    | end
    | 
    | # given a struct from analyze_touchpoints_only(), calculate the points
    | # for left, for extended
    | def calculate_DOtA_points_left_extended(struct1, listleans, chamferover, tcp_pose_top):
    |     # get the stuff from the struct
    |     pointintersect = struct1[0]
    |     heading1 = struct1[1]
    |     heading2 = struct1[2]
    |     heading3 = struct1[3]
    |     l1delxunit = struct1[4]
    |     l1delyunit = struct1[5]
    |     l2delxunit = struct1[6]
    |     l2delyunit = struct1[7]
    | 
    |     # FIND THE POINTS ON THE LINES OF THE FIRST TURN PATH
    |     # find locations 8 inches away from  intersect point
    |     # CONST
    |     # welddistance1 = 8 # vertical weld distance
    |     welddistance2 = 6 # first path second leg
    |     welddistance3 = 8 # second path second leg
    |     zup = .375
    |     # inches
    |     # wd1 = welddistance1 * 25.4 / 1000
    |     wd2 = welddistance2 * 25.4 / 1000
    |     wd3 = welddistance3 * 25.4 / 1000
    |     zup = zup * 25.4 / 1000
    |     chamferovermm =  chamferover * 25.4 / 1000
    | 
    |     # weld distance is the distance that it will weld. this will make it start at the z height that the user specified
    |     wd1 = tcp_pose_top[2] - pointintersect[2] - zup
    | 
    |     x = pointintersect[0] + l2delxunit * chamferovermm
    |     y = pointintersect[1] + l2delyunit * chamferovermm
    |     z = pointintersect[2] + zup
    | 
    |     #apply actual rxryrz to points
    |     # convert the headings to rxryrz and insert those values into the relevant points
    |     rxryrz = convert_heading_to_axang_preheatdown(heading3)
    |     rx = rxryrz[0]
    |     ry = rxryrz[1]
    |     rz = rxryrz[2]
    | 
    |     point1 = p[x + wd1*listleans[0], y + wd1*listleans[1], z + wd1, rx, ry, rz]
    |     point2 = p[x, y, z, rx, ry, rz]
    | 
    |     # convert the headings to rxryrz and insert those values into the relevant points
    |     rxryrz = convert_heading_to_axang(heading3)
    |     rx = rxryrz[0]
    |     ry = rxryrz[1]
    |     rz = rxryrz[2]
    | 
    |     point4 = p[x, y, z, rx, ry, rz]
    |     x = x + l2delxunit * wd2
    |     y = y + l2delyunit * wd2
    |     point5 = p[x, y, z, rx, ry, rz]
    | 
    |     # FIND THE POINTS ON THE LINES OF THE SECOND AROUND PATH
    |     roundoverdistance = 0.05
    |     rod = roundoverdistance * 25.4 / 1000
    | 
    |     # now we have the unit vector. extend the weld distance from the intersection
    |     x = pointintersect[0] + l2delxunit * chamferovermm
    |     y = pointintersect[1] + l2delyunit * chamferovermm
    |     # convert the headings to rxryrz and insert those values into the relevant points
    |     rxryrz = convert_heading_to_axang_ccw(heading3)
    |     rx = rxryrz[0]
    |     ry = rxryrz[1]
    |     rz = rxryrz[2]
    |     point_1 = p[x, y, z, rx, ry, rz]
    | 
    |     x = pointintersect[0] + l2delxunit * rod
    |     y = pointintersect[1] + l2delyunit * rod
    |     point_2 = p[x, y, z, rx, ry, rz]
    | 
    |     # convert the headings to rxryrz and insert those values into the relevant points
    |     rxryrz = convert_heading_to_axang_ccw(heading1)
    |     rx = rxryrz[0]
    |     ry = rxryrz[1]
    |     rz = rxryrz[2]
    | 
    |     x = pointintersect[0] + l1delxunit * rod
    |     y = pointintersect[1] + l1delyunit * rod
    |     point_4 = p[x, y, z, rx, ry, rz]
    | 
    |     # extend the weld distance from the intersection
    |     valid1 = True
    |     # start with the seed
    |     x = pointintersect[0] + l1delxunit * wd3
    |     y = pointintersect[1] + l1delyunit * wd3
    |     point_5 = p[x, y, z, rx, ry, rz]
    |     seed = p[x, y, z, rx, ry, rz]
    |     valid1 = get_inverse_kin_has_solution(seed)
    |     # define the increment
    |     increment = 1.0 # inches
    |     increment = increment * 25.4 / 1000 # meters
    |     while valid1 == True:
    |         wd3 = wd3 + increment
    |         x = pointintersect[0] + l1delxunit * wd3
    |         y = pointintersect[1] + l1delyunit * wd3
    |         seed = p[x, y, z, rx, ry, rz]
    |         valid1 = get_inverse_kin_has_solution(seed)
    |     end
    |     # move back 1 to get the highest valid wd3
    |     # move back 3 to get the third highest valid wd3
    |     wd3 = wd3 - (3.0 * increment)
    |     x = pointintersect[0] + l1delxunit * wd3
    |     y = pointintersect[1] + l1delyunit * wd3
    |     point_5 = p[x, y, z, rx, ry, rz]
    | 
    |     #FIND POINT 3
    |     # by calling analyze_touchpoints()
    |     atret = analyze_touchpoints(point_2, point_1, point_4, point_5, pointintersect)
    |     point_3 = atret[5]
    |     #point 3 will not have the correct rxryrz though because now the gun needs to be face up
    |     rxryrz = convert_heading_to_axang_ccw(heading2)
    |     rx = rxryrz[0]
    |     ry = rxryrz[1]
    |     rz = rxryrz[2]
    |     point_3 = p[point_3[0], point_3[1], point_3[2], rx, ry, rz]
    | 
    |     struct2 = struct(point1=point1, point2=point2, point4=point4, point5=point5, point_1=point_1, point_2=point_2, point_3=point_3, point_4=point_4, point_5=point_5)
    |     return struct2
    | end
    | 
    | # this function analyzes the vertical points
    | # calculates the slope of the edge in question
    | # specifically, for each inch up in the z direction, what is the change in x and change in y direction
    | # returns a list of [nx, ny]
    | def analyze_vertical_touchpoints(p11, p12, p13, p21, p22, p23, p3):
    |     # first, find the equations of the planes from the 6 points
    |     plane1 = findplane(p11, p12, p13)
    |     plane2 = findplane(p21, p22, p23)
    |     # Find the Direction Vector of the Line: The direction vector d of the line of intersection can be found by taking the cross product of the normal vectors of each plane (a, b, and c)
    |     nx = plane1[1]*plane2[2] - plane1[2]*plane2[1]
    |     ny = plane1[2]*plane2[0] - plane1[0]*plane2[2]
    |     nz = plane1[0]*plane2[1] - plane1[1]*plane2[0]
    |     # normalize the vector so the z length is 1
    |     multiplier = 1 / nz
    |     nx = nx * multiplier
    |     ny = ny * multiplier
    |     nz = nz * multiplier # should become equal to 1
    |     ret = [nx, ny]
    |     return ret
    | end
    | 
    | # given 3 points, this finds the plane and its equation
    | # rereturns ax + by + cz + d = 0 in a list of [a, b, c, d]
    | def findplane(p11, p12, p13):
    |     # extract coordinates
    |     x1 = p11[0]
    |     y1 = p11[1]
    |     z1 = p11[2]
    |     x2 = p12[0]
    |     y2 = p12[1]
    |     z2 = p12[2]
    |     x3 = p13[0]
    |     y3 = p13[1]
    |     z3 = p13[2]
    |     # create vectors from the points
    |     v1x = x2-x1
    |     v1y = y2-y1
    |     v1z = z2-z1
    |     v2x = x3-x1
    |     v2y = y3-y1
    |     v2z = z3-z1
    |     #calculate the normal vector using the cross product
    |     nx = v1y*v2z - v1z*v2y # i component
    |     ny = v1z*v2x - v1x*v2z # j component
    |     nz = v1x*v2y - v1y*v2x # k component
    |     # calculate d in the plane equation
    |     d = -1 * (nx*x1 + ny*y1 + nz*z1)
    |     ret = [nx, ny, nz, d]
    |     return ret
    | end
    | 
    | # given a heading, (ccw from +x axis), find the mx+b slope
    | # fails if exactly vertical
    | def get_slope_from_heading(heading):
    |     return tan(heading)
    | end
    | 
    | 
    | 
    | # this function finds the points (and rxryrz) of the 2 points (start and end) of vertical weld section
    | def find_vertical_points(pointintersect, l1delxunit, l1delyunit, l2delxunit, l2delyunit, offset, wd, heading1, heading3):
    | 
    |   # find right side stuff
    |   # find the point in 3d space that is .375 up and .375 over
    |   x = pointintersect[0] + l1delxunit * offset
    |   y = pointintersect[1] + l1delyunit * offset
    |   z = pointintersect[2] + offset
    |   # find rxryrz
    |   rxryrz = convert_heading_to_axang_preheatup(heading1)
    |   rx = rxryrz[0]
    |   ry = rxryrz[1]
    |   rz = rxryrz[2]
    |   path2r1 = p[x, y, z, rx, ry, rz]
    |   path2r2 = p[x, y, z + wd, rx, ry, rz]
    | 
    |   # find left side
    |   # find the point in 3d space that is .375 up and .375 over
    |   x = pointintersect[0] + l2delxunit * offset
    |   y = pointintersect[1] + l2delyunit * offset
    |   z = pointintersect[2] + offset
    |   # find rxryrz
    |   rxryrz = convert_heading_to_axang_preheatup(heading3)
    |   rx = rxryrz[0]
    |   ry = rxryrz[1]
    |   rz = rxryrz[2]
    |   path2l1 = p[x, y, z, rx, ry, rz]
    |   path2l2 = p[x, y, z + wd, rx, ry, rz]
    | 
    |   ret = struct(path2r1=path2r1, path2r2=path2r2, path2l1=path2l1, path2l2=path2l2)
    |   return ret
    | end
    | 
    | # this function converts a unit vector to its heading angle ccw from x+ axis
    | # takes uvx and uvy
    | # returns heading in radians
    | def convert_uv_to_heading(uvx, uvy):
    |   baseang = atan(uvy/uvx)
    |   if uvx < 0:
    |     ang = baseang + pi
    |   elif uvy < 0:
    |     ang = baseang + pi * 2
    |   else:
    |     ang = baseang
    |   end
    |   return ang
    | end
    | 
    | # this function finds the equation of a line, perpendicular to a given line, and going through a given point
    | # takes 3 arguments: m (the original line's slope), x (point's x coord), y (point's y coord). the b of the original line is not needed
    | # returns a list of [m,b] (the slope and intercept of the new line)
    | def find_perpendicular_line(origm, x, y):
    |   m = (1/origm) * -1
    |   b = y - m*x
    |   ret = [m, b]
    |   return ret
    | end
    | 
    | # this function finds the intersection point between two lines in the xy plane
    | # takes 4 arguments: m1, b1, m2, b2
    | # returns a list of [x,y] (the point of intersection)
    | def find_intersection(m1, b1, m2, b2):
    |   # m1x+b1 = m2x+b2
    |   # m1x - m2x = b2 - b1
    |   # x = (b2-b1) / (m1-m2)
    |   x = (b2-b1) / (m1-m2)
    |   y = m1 * x + b1
    |   ret = [x, y]
    |   return ret
    | end
    | 
    | # this function finds the distance between 2 points in 3d space
    | # it takes 6 arguments: x1, y1, z1, x2, y2, z2
    | # it returns a distance
    | def distance_between(x1, y1, z1, x2, y2, z2):
    |   distsquared = (x2-x1)*(x2-x1)+(y2-y1)*(y2-y1)+(z2-z1)*(z2-z1)
    |   dist = sqrt(distsquared)
    |   return dist
    | end
    | 
    | # this function takes a point, a unit vector, and a distance, and adds the distance to the point in the direction of the unit vector (3d space)
    | # it returns a point as a list of coordinates
    | def add_vectordistance_to_point(xi, yi, zi, uvx, uvy, uvz, delta):
    |   xf = xi + uvx * delta
    |   yf = yi + uvy * delta
    |   zf = zi + uvz * delta
    |   ret = [xf, yf, zf]
    |   return ret
    | end
    | 
    | # this function converts a heading (ccw radians from the positive x axis) into rxryrz to be put into a point p[]
    | # this will point the gun in this heading with the bottom side of the gun facing up.
    | # the values used in this program were calculated by doing rotation matrix math in the file on WI-CALVINB10 C. Documents. Theory for converting rotations into axis angle representations
    | def convert_heading_to_axang(heading):
    |  axisxraw = -1 * sin(heading)
    |  axisyraw = cos(heading) + 1
    |  axiszraw = sin(heading)
    | 
    |  magnitude = sqrt(axisxraw*axisxraw + axisyraw*axisyraw + axiszraw*axiszraw)
    | 
    |  axisxunit = axisxraw / magnitude
    |  axisyunit = axisyraw / magnitude
    |  axiszunit = axiszraw / magnitude
    | 
    |  angle = acos( (cos(heading) - 1) / 2 )
    | 
    |  rxout = axisxunit * angle
    |  ryout = axisyunit * angle
    |  rzout = axiszunit * angle
    | 
    |  return [rxout, ryout, rzout]
    | end
    | 
    | # this function converts a heading (ccw radians from the positive x axis) into rxryrz to be put into a point p[]
    | # this will point the gun in this heading with the preheat side of the gun tip facing up. Used for welding in a vertical path.
    | # the values used in this program were calculated by doing rotation matrix math in the file on WI-CALVINB10 C. Documents. Theory for converting rotations into axis angle representations
    | def convert_heading_to_axang_preheatup(heading):
    |  axisxraw = -sin(heading) + 1
    |  axisyraw = cos(heading)
    |  axiszraw = cos(heading)
    | 
    |  magnitude = sqrt(axisxraw*axisxraw + axisyraw*axisyraw + axiszraw*axiszraw)
    | 
    |  axisxunit = axisxraw / magnitude
    |  axisyunit = axisyraw / magnitude
    |  axiszunit = axiszraw / magnitude
    | 
    |  angle = acos( (-sin(heading) - 1) / 2 )
    | 
    |  rxout = axisxunit * angle
    |  ryout = axisyunit * angle
    |  rzout = axiszunit * angle
    | 
    |  return [rxout, ryout, rzout]
    | end
    | 
    | # this function converts a heading (ccw radians from the positive x axis) into rxryrz to be put into a point p[]
    | # this will point the gun in this heading with the preheat side of the gun tip facing down. Used for welding in a vertical path downwards.
    | # the values used in this program were calculated by doing rotation matrix math in the file on WI-CALVINB10 C. Documents. Theory for converting rotations into axis angle representations
    | def convert_heading_to_axang_preheatdown(heading):
    |  axisxraw = -sin(heading) - 1
    |  axisyraw = cos(heading)
    |  axiszraw = -cos(heading)
    | 
    |  magnitude = sqrt(axisxraw*axisxraw + axisyraw*axisyraw + axiszraw*axiszraw)
    | 
    |  axisxunit = axisxraw / magnitude
    |  axisyunit = axisyraw / magnitude
    |  axiszunit = axiszraw / magnitude
    | 
    |  angle = acos( (sin(heading) - 1) / 2 )
    | 
    |  rxout = axisxunit * angle
    |  ryout = axisyunit * angle
    |  rzout = axiszunit * angle
    | 
    |  return [rxout, ryout, rzout]
    | end
    | 
    | # this function converts a heading (ccw radians from the positive x axis) into rxryrz to be put into a point p[]
    | # this will point the gun in this heading with the preheat side of the gun tip facing right. Used for welding counterclockwise around the box.
    | # the values used in this program were calculated by doing rotation matrix math in the file on WI-CALVINB10 C. Documents. Theory for converting rotations into axis angle representations
    | def convert_heading_to_axang_ccw(heading):
    |  axisxraw = -sin(heading)
    |  axisyraw = cos(heading) - 1
    |  axiszraw = -sin(heading)
    | 
    |  magnitude = sqrt(axisxraw*axisxraw + axisyraw*axisyraw + axiszraw*axiszraw)
    | 
    |  axisxunit = axisxraw / magnitude
    |  axisyunit = axisyraw / magnitude
    |  axiszunit = axiszraw / magnitude
    | 
    |  angle = acos( (-cos(heading) - 1) / 2 )
    | 
    |  rxout = axisxunit * angle
    |  ryout = axisyunit * angle
    |  rzout = axiszunit * angle
    | 
    |  return [rxout, ryout, rzout]
    | end
    | 
    | # this function takes two rotation matrices, and multiplies them together, returning one matrix.
    | # all matrices are in the form of a list.
    | # all matrix values have constant values (no variables)
    | def multiply_matrix(matrix1, matrix2):
    |     # retrieve values
    |     a11 = matrix1[0]
    |     a12 = matrix1[1]
    |     a13 = matrix1[2]
    |     a21 = matrix1[3]
    |     a22 = matrix1[4]
    |     a23 = matrix1[5]
    |     a31 = matrix1[6]
    |     a32 = matrix1[7]
    |     a33 = matrix1[8]
    |     b11 = matrix2[0]
    |     b12 = matrix2[1]
    |     b13 = matrix2[2]
    |     b21 = matrix2[3]
    |     b22 = matrix2[4]
    |     b23 = matrix2[5]
    |     b31 = matrix2[6]
    |     b32 = matrix2[7]
    |     b33 = matrix2[8]
    |     #calculate c values
    |     c11 = a11*b11 + a12*b21 + a13*b31
    |     c12 = a11*b12 + a12*b22 + a13*b32
    |     c13 = a11*b13 + a12*b23 + a13*b33
    |     c21 = a21*b11 + a22*b21 + a23*b31
    |     c22 = a21*b12 + a22*b22 + a23*b32
    |     c23 = a21*b13 + a22*b23 + a23*b33
    |     c31 = a31*b11 + a32*b21 + a33*b31
    |     c32 = a31*b12 + a32*b22 + a33*b32
    |     c33 = a31*b13 + a32*b23 + a33*b33
    |     # return resulting matrix
    |     ret = [c11, c12, c13, c21, c22, c23, c31, c32, c33]
    |     return ret
    | end
    | 
    | # this function converts a matrix to axis angle representations
    | # this matrix is usually a resulting matrix (result of matrix multiplication) in normal use, given as a list
    | # returns a list of [rx,ry,rz]
    | def convert_matrix_to_axang(matrix1):
    |     # retrieve values
    |     a11 = matrix1[0]
    |     a12 = matrix1[1]
    |     a13 = matrix1[2]
    |     a21 = matrix1[3]
    |     a22 = matrix1[4]
    |     a23 = matrix1[5]
    |     a31 = matrix1[6]
    |     a32 = matrix1[7]
    |     a33 = matrix1[8]
    | 
    |     # First Half: find the angle
    |     # find the trace
    |     # using the formula: trace = a11 + a22 + a33
    |     trace = a11 + a22 + a33
    |     # find the angle using the formula: trace(matrix) = 1 + 2 cos(angle)
    |     angle = acos((trace - 1.0)/2.0)
    | 
    |     # Second Half: calculate the rotation axis
    |     axisxraw = a32 - a23
    |     axisyraw = a13 - a31
    |     axiszraw = a21 - a12
    |     # normalize axis
    |     magnitude = sqrt(axisxraw*axisxraw + axisyraw*axisyraw + axiszraw*axiszraw)
    |     axisxunit = axisxraw / magnitude
    |     axisyunit = axisyraw / magnitude
    |     axiszunit = axiszraw / magnitude
    | 
    |     # combine axis and angle into rxryrz representation
    |     rxout = axisxunit * angle
    |     ryout = axisyunit * angle
    |     rzout = axiszunit * angle
    |     return [rxout, ryout, rzout]
    | end
    | 
    | # this function takes a rotation and calculates the corresponding rotation matrix
    | # input is (axis, direction, angle in radians)
    | # example is ("x", 1, pi/6) = a 30 degree turn around the x axis in the positive direction (right hand rule)
    | # returns a matrix (a list of 9 values)
    | def get_rotation_matrix_from_description(axis, direction, angle):
    |     # get the angle
    |     a = angle * direction
    |     # get the axis
    |     if axis == "x" or axis == "X":
    |         matrix = [1, 0, 0, 0, cos(a), -1 * sin(a), 0, sin(a), cos(a)]
    |         return matrix
    |     end
    |     if axis == "y" or axis == "Y":
    |         matrix = [cos(a), 0, sin(a), 0, 1, 0, -1*sin(a), 0, cos(a)]
    |         return matrix
    |     end
    |     if axis == "z" or axis == "Z":
    |         matrix = [cos(a), -1*sin(a), 0, sin(a), cos(a), 0, 0, 0, 1]
    |         return matrix
    |     end
    |     # bad
    |     popuptext = "Error in get_rotation_matrix_from_description. "
    |     # infinite loop
    |     while 1==1:
    |       popup(popuptext, title="Code Error",blocking=True)
    |     end
    | end
    | 
    | # this function is for getting the points along the path of the corner homing 45
    | # point0 is the point where they touched
    | def get_corner_homing_45_pathpoints(point0, pointtop = p[0,0,0,0,0,0]):
    |   p0x = point0[0]
    |   p0y = point0[1]
    |   p0z = point0[2]
    |   p0rx = point0[3]
    |   p0ry = point0[4]
    |   p0rz = point0[5]
    | 
    |   #constants
    |   #distances of how far away from point the touchpoints are
    |   d0 = 0.10 # how far from the box to retreat and approach
    |   d1 = 0.03 # first distance from init point
    |   d2 = 0.15 # second distance from init point
    |   d3 = 0.125 #vertical distance from first point
    |   sqrt2 = 0.707106781 # 1/sqrt(2) , the inverse of the sqrt(2)
    | 
    |   ph1 = p[p0x + d0, p0y, p0z + d1, p0rx, p0ry, p0rz] #approach point for turn
    | 
    |   ph2 = p[p0x+d0-d0*0.5-sqrt2*d1, p0y+d0*0.5+sqrt2*d1, p0z+d1, 1.446, -0.8, -0.733]
    |   ph3 = p[p0x+d0-d0*0.5-sqrt2*d2, p0y+d0*0.5+sqrt2*d2, p0z+d1, 1.446, -0.8, -0.733]
    |   ph4 = p[p0x+d0-d0*0.5-sqrt2*d1, p0y-d0*0.5-sqrt2*d1, p0z+d1, 0.626, -1.993, -1.813]
    |   ph5 = p[p0x+d0-d0*0.5-sqrt2*d2, p0y-d0*0.5-sqrt2*d2, p0z+d1, 0.626, -1.993, -1.813]
    | 
    |   # go back to ph1
    |   ph6 = p[p0x + d0, p0y, p0z -0.05, 0, 0, 0] # approach point for under turn
    |   # moveL from ph1 to ph6
    |   ph7 = p[p0x-d1, p0y, p0z-0.05, 0, 0, 0]
    | 
    |   # add the vertical touch points
    |   if pointtop[2] == 0:
    |     ph2up = p[ph2[0], ph2[1], ph2[2]+d3, ph2[3], ph2[4], ph2[5]]
    |     ph4up = p[ph4[0], ph4[1], ph4[2]+d3, ph4[3], ph4[4], ph4[5]]
    |   else:
    |     ph2up = p[ph2[0], ph2[1], pointtop[2], ph2[3], ph2[4], ph2[5]]
    |     ph4up = p[ph4[0], ph4[1], pointtop[2], ph4[3], ph4[4], ph4[5]]
    |   end
    |   ret = struct(ph1=ph1, ph2=ph2, ph3=ph3, ph4=ph4, ph5=ph5, ph6=ph6, ph7=ph7, ph2up=ph2up, ph4up=ph4up)
    |   is_robot_at_reachable_spot(point0, ret)
    |   return ret
    | end
    | 
    | # this function checks whether the touchpoints are reachable AKA is the robot positioned in the right spot
    | # if everything looks good, it continues.
    | # if it detects a problem, it infinite loops a popup
    | def is_robot_at_reachable_spot(point0, struct_touchpoints):
    |   # first, check whether the corner is too low to the ground that the bottom homing will hit the ground (z < -350)
    |   lc_height = get_lift_column_height_condensed()
    |   # total height = zeroed lift column height (41.25 inches) (1.04775 m) plus lift column height plus robot relative height
    |   totalheight = 1.04775 + lc_height + point0[2]
    |   if totalheight < 1.04775 - 0.350:
    |     # bad
    |     popuptext = "Tank Corner is too low to the ground. Collisions will occur. Stop Program and raise tank. "
    |     # infinite loop
    |     while 1==1:
    |       popup(popuptext, title="Robot Positioning Warning",blocking=True)
    |     end
    |   end
    | 
    | 
    | 
    |   # next, check whether the touchpoints are reachable
    |   allvalid = check_structofpoints_validity(struct_touchpoints)
    |   if not allvalid:
    | 
    |     # then unreachable
    |     # generate message
    |     listproblems = ""
    |     listnames = ["ph1", "ph2", "ph3", "ph4", "ph5", "ph6", "ph7", "ph2up", "ph4up"]
    |     i = 0
    |     structlength = 9
    |     while i < structlength:
    |       curr = struct_touchpoints[i]
    |       valid = get_inverse_kin_has_solution(curr)
    |       if not valid:
    |         listproblems = listproblems + listnames[i]
    |       end
    |       i = i + 1
    |     end
    |     # display
    |     popuptext = "Robot is too far from tank corner. Cannot reach some necessary positions. Stop Program and move robot closer. " + listproblems
    |     # infinite loop
    |     while 1==1:
    |       popup(popuptext, title="Robot Positioning Warning",blocking=True)
    |     end
    |   end
    | 
    | end
    | 
    | # this function takes a struct of points as an argument, and checks whether every point in the list is reachable using get_inverse_kin_has_solution()
    | # this function does NOT check for weird twists or joint limits
    | # inputstruct must contain only points
    | # it returns true if all points are valid. it returns false if any points are valid
    | # a list of length 0 indicates that all points are valid
    | def check_structofpoints_validity(inputstruct):
    |   # next, check whether the touchpoints are reachable
    |   structlength = length(inputstruct)
    |   i = 0
    |   allvalid = True
    |   while i < structlength:
    |     curr = inputstruct[i]
    |     valid = get_inverse_kin_has_solution(curr)
    |     if not valid:
    |       return False
    |     end
    |     i = i + 1
    |   end
    |   return True
    | end
    | 
    | # checks the validity of all points during a left weld
    | def check_validity_left(struct1, struct2):
    |   #first, check whether robot is too close
    |   pointintersect = struct1[0]
    |   # next, check if the corner is too close to the robot to do a left around weld (complex but approximately X > -1300)
    |   # if y < 0, then x < -1300. if y < 480, then y > (1300+x)*8. if y > 480, then y > (1235+x)*4 + 500
    |   toocloseleftweld = False
    |   if pointintersect[1] < 0:
    |     if pointintersect[0] > -1.300:
    |       toocloseleftweld = True
    |     end
    |   elif pointintersect[1] < 0.480:
    |     if pointintersect[1] < (1.300 + pointintersect[0])*8:
    |       toocloseleftweld = True
    |     end
    |   else:
    |     if pointintersect[1] < (1.235 + pointintersect[0])*4 + 0.500:
    |       toocloseleftweld = True
    |     end
    |   end
    |   if toocloseleftweld:
    |     # bad
    |     popuptext = "Robot is too close to tank corner. Collisions may occur. Stop Program and move robot farther. "
    |     # infinite loop
    |     while 1==1:
    |       popup(popuptext, title="Robot Positioning Warning",blocking=True)
    |     end
    |   end
    | 
    |   #next, check whether all the points in the weldpath are valid
    |   structlength = 9
    |   i = 0
    |   allvalid = True
    |   listproblems = ""
    |   listnames = ["point1", "point2", "point4", "point5", "point_1", "point_2", "point_3", "point_4", "point_5"]
    |   while i < structlength:
    |     curr = struct2[i]
    |     valid = get_inverse_kin_has_solution(curr)
    |     if not valid:
    |       allvalid = False
    |       listproblems = listproblems + listnames[i]
    |     end
    |     i = i + 1
    |   end
    | 
    |   if not allvalid:
    |     # display
    |     popuptext = "Robot is too far from tank corner. Cannot reach some necessary positions. Stop Program and move robot closer. " + listproblems
    |     # infinite loop
    |     while 1==1:
    |       popup(popuptext, title="Robot Positioning Warning",blocking=True)
    |     end
    |   end
    | 
    |   # check whether the path involves weird turns or joint limits. currently just checks the first position
    |   p_prev = [-0.021118, -1.26292, 2.43578, 5.07088, -2.29912, 1.53362] #last point of left weld prerotate
    |   joints_1 = get_inverse_kin(struct2[0], p_prev) # struct2[0] is point1
    |   allGood = True
    |   i = 0
    |   structlength = 6
    |   while i < structlength:
    |     joint_curr = joints_1[i]
    |     # check for anything that exceeds joint limits
    |     degreesmax = 360 * pi / 180
    |     if joint_curr > degreesmax or joint_curr < degreesmax * -1:
    |       allGood = False
    |     end
    |     # check for anything that is significantly different than the aligned approach. could indicate a twist is needed. we dont want that
    |     maxdifference = 150 * pi / 180
    |     difference = joint_curr - p_prev[i]
    |     if difference > maxdifference or difference * -1 > maxdifference:
    |       allGood = False
    |     end
    |     i = i + 1
    |   end
    | 
    |   if not allGood:
    |     # display
    |     popuptext = "Top of Weld is too high above robot. Cannot reach some necessary positions. Stop Program and try again with a lower top point. "
    |     # infinite loop
    |     while 1==1:
    |       popup(popuptext, title="Robot Positioning Warning",blocking=True)
    |     end
    |   end
    | 
    | end
    | 
    | # checks the validity of all points during a right weld
    | def check_validity_right(struct1, struct2):
    |   # first, check whether the right pivot will bonk itself
    |   pointintersect = struct1[0]
    |   heading1 = struct1[1] # this is the direction that the welder will face when doing the right side of the box
    | 
    |   #first, check whether the heading is just too far offset
    |   # more than 15 degrees off of 45 is too much
    |   # normal heading is 216 degrees
    |   #201 degrees to 231 degrees
    |   heading1degrees = heading1 * 180 / pi
    |   if heading1degrees < 201 or heading1degrees > 231 :
    |     # then out of range
    |     popuptext = "Robot is not aligned at a 45 degree angle of corner (15 degree leeway). Collisions may occur. Stop Program and align robot. heading1degrees=" + str_cat("",heading1degrees)
    |     # infinite loop
    |     while 1==1:
    |       popup(popuptext, title="Robot Positioning Warning",blocking=True)
    |     end
    |   end
    | 
    |   #TODO: add the checks for whether x is too close, given the heading
    |   # add checks for whether x is too close, given the heading
    |   # different equations for whether heading offset > 5 degrees or less (inc. negative)
    |   headingoffset = heading1degrees - 216
    |   if headingoffset < 5:
    |     # then calculate a and b
    |     a = 0.4584 + -0.02369 * headingoffset
    |     b = (-1151.4 + 13.83 * headingoffset) / 1000
    |     # check whether x > a*y+b
    |     if pointintersect[0] > a * pointintersect[1] + b:
    |       # bad
    |       popuptext = "Robot is too close to tank corner or not at the right angle. Collisions may occur. Stop Program and align robot. "
    |       # infinite loop
    |       while 1==1:
    |         popup(popuptext, title="Robot Positioning Warning",blocking=True)
    |       end
    |     end
    |   else:
    |     # headingoffset > 5 degrees
    |     if pointintersect[1] < 0:
    |       if pointintersect[0] > -1150.0 / 1000.0:
    |         #bad
    |         popuptext = "Robot is too close to tank corner. Collisions may occur. Stop Program and align robot. "
    |         # infinite loop
    |         while 1==1:
    |           popup(popuptext, title="Robot Positioning Warning",blocking=True)
    |         end
    |       end
    |     else:
    |       # if x > .7736 y - 1101.9 then bad
    |       if pointintersect[0] > 0.7736 * pointintersect[1] - 1101.9 / 1000:
    |         popuptext = "Robot is too close to tank corner. Collisions may occur. Stop Program and align robot. "
    |         # infinite loop
    |         while 1==1:
    |           popup(popuptext, title="Robot Positioning Warning",blocking=True)
    |         end
    |       end
    |     end
    |   end
    | 
    |   #next, check whether all the points in the weldpath are valid
    |   structlength = 9
    |   i = 0
    |   allvalid = True
    |   listproblems = ""
    |   listnames = ["point1", "point2", "point4", "point5", "point_1", "point_2", "point_3", "point_4", "point_5"]
    |   while i < structlength:
    |     curr = struct2[i]
    |     valid = get_inverse_kin_has_solution(curr)
    |     if not valid:
    |       allvalid = False
    |       listproblems = listproblems + listnames[i]
    |     end
    |     i = i + 1
    |   end
    | 
    |   if not allvalid:
    |     # display
    |     popuptext = "Robot is too far from tank corner. Cannot reach some necessary positions. Stop Program and move robot closer. " + listproblems
    |     # infinite loop
    |     while 1==1:
    |       popup(popuptext, title="Robot Positioning Warning",blocking=True)
    |     end
    |   end
    | 
    |   # check whether the path involves weird turns or joint limits. currently just checks the first position
    |   p_prev = [-1.13307, -1.48911, 2.84785, 4.92357, -4.89059, 1.57184] #last point of right weld prerotate
    |   joints_1 = get_inverse_kin(struct2[0], p_prev) # struct2[0] is point1
    |   allGood = True
    |   i = 0
    |   structlength = 6
    |   while i < structlength:
    |     joint_curr = joints_1[i]
    |     # check for anything that exceeds joint limits
    |     degreesmax = 360 * pi / 180
    |     if joint_curr > degreesmax or joint_curr < degreesmax * -1:
    |       allGood = False
    |     end
    |     # check for anything that is significantly different than the aligned approach. could indicate a twist is needed. we dont want that
    |     maxdifference = 150 * pi / 180
    |     difference = joint_curr - p_prev[i]
    |     if difference > maxdifference or difference * -1 > maxdifference:
    |       allGood = False
    |     end
    |     i = i + 1
    |   end
    | 
    |   if not allGood:
    |     # display
    |     popuptext = "Top of Weld is too high above robot. Cannot reach some necessary positions. Stop Program and try again with a lower top point. "
    |     # infinite loop
    |     while 1==1:
    |       popup(popuptext, title="Robot Positioning Warning",blocking=True)
    |     end
    |   end
    | end
    | 
    | # this function sends a signal to turn extrusion on
    | def turn_extrusion_on():
    |   # flush the channel
    |   resp0 = send_serial_signal(["u", "r", "?"])
    |   # send the signal
    |   resp1 = send_serial_signal(["u", "R", "1"])
    |   # if resp <> "uR1"
    |   if resp1 != [252,82,49]:
    |     # turn off extrusion and heating. inform calvin
    |     resp2 = send_serial_signal(["u", "R", "0"])
    |     resp3 = send_serial_signal(["u", "H", "0"])
    |     popuptext = "Error code encountered while trying to start extrusion. Find Calvin. "
    |     while 1==1:
    |       popup(popuptext, title="Extrusion Error Code",blocking=True)
    |       popup(resp1, blocking=True)
    |     end
    |   end
    | end
    | 
    | # this function sends a signal and receives a response
    | # signal is a list of 3 strings, 1 character each. first is u. second is the next character. third is final character
    | def send_serial_signal(signal):
    |   signal2char = signal[1]
    |   signal3char = signal[2]
    |   listsignal = [252, get_corr_number(signal2char), get_corr_number(signal3char)]
    |   resp1 = WTSerialBridge.send_command("/dev/ttyUSB0",1200, 8, "None", "One", "None", 1000, "None", "None", listsignal, True)
    |   return resp1
    | end
    | 
    | # this function converts a letter into its ascii number
    | def get_corr_number(letter):
    |   if letter == "A":
    |     return 65
    |   elif letter == "H":
    |     return 72
    |   elif letter == "R":
    |     return 82
    |   elif letter == "M":
    |     return 77
    |   elif letter == "E":
    |     return 69
    |   elif letter == "a":
    |     return 97
    |   elif letter == "b":
    |     return 98
    |   elif letter == "h":
    |     return 104
    |   elif letter == "r":
    |     return 114
    |   elif letter == "s":
    |     return 115
    |   elif letter == "m":
    |     return 109
    |   elif letter == "0":
    |     return 48
    |   elif letter == "1":
    |     return 49
    |   elif letter == "2":
    |     return 50
    |   elif letter == "3":
    |     return 51
    |   elif letter == "4":
    |     return 52
    |   elif letter == "5":
    |     return 53
    |   elif letter == "6":
    |     return 54
    |   elif letter == "7":
    |     return 55
    |   elif letter == "8":
    |     return 56
    |   elif letter == "9":
    |     return 57
    |   elif letter == "?":
    |     return 63
    |   end
    | end
    | 
    | # this function checks whether the welder is in the ready state.
    | # to be called at the beginning of Main Program
    | def welder_state_ready():
    |   # flush the channel
    |   resp0 = send_serial_signal(["u", "s", "?"])
    |   # send the signal
    |   resp1 = send_serial_signal(["u", "s", "?"])
    |   # if resp1 == [252,115,49] (us1) then it is ready. otherwise, it is not
    |   if resp1 != [252,115,49]:
    |     popuptext = "Welder is not ready for extrusion. Follow the instructions to start heating welder. "
    |     while 1==1:
    |       popup(popuptext, title="Welder Not Ready",blocking=True)
    |     end
    |   end
    | 
    | end
    | 
    | def get_lift_column_height():
    |   # begin: URCap Program Node
    |   #   Source: MachineLogic for Universal Robots, 3.1.7, Vention Inc.
    |   #   Type: MachineLogic for Universal Robots
    |   #$ 5 "MachineLogic Get Position"
    |   while isVentionMovementBusyMachineMotion1==True:
    |     sleep(0.05)
    |   end
    |   if(isVentionMovementBusyMachineMotion1 == False):
    |     isVentionMovementBusyMachineMotion1 = True
    |     socket_send_string("estop/status;", "MachineMotion1")
    |     temp_estop_var_vention = socket_read_string("MachineMotion1",timeout=15)
    |     while(temp_estop_var_vention=="estop/status true"):
    |       if temp_estop_var_vention=="estop/status true":
    |         sendStringWithTimeout("estop/systemreset/request","Ack estop/systemreset/request;","MachineMotion1")
    |       end
    |       socket_send_string("estop/status;", "MachineMotion1")
    |       temp_estop_var_vention = socket_read_string("MachineMotion1",timeout=15)
    |       if temp_estop_var_vention=="estop/status true":
    |         popup("MachineMotion in estop, make sure you have all emergency modules released manually. If you continue the system will try to reset MachineMotion automatically.",blocking=True)
    |       end
    |     end
    |   else:
    |     popup("resource is being used already: MachineMotion1")
    |     halt
    |   end
    |   socket_send_string("GET im_get_controller_pos_axis_1;", "MachineMotion1")
    |   temp_drive = socket_read_ascii_float(1, "MachineMotion1",timeout=15)
    |   global var_1 = temp_drive[1]
    |   isVentionMovementBusyMachineMotion1 = False
    |   sleep(0.03)
    |   # end: URCap Program Node
    | end
    | 
    | def get_lift_column_height_condensed():
    |   socket_send_string("GET im_get_controller_pos_axis_1;", "MachineMotion1")
    |   temp_drive = socket_read_ascii_float(1, "MachineMotion1",timeout=15)
    |   ret = temp_drive[1]
    |   return ret
    | end
  Script: welder_state_ready()
  leftchoice :=  (valueSource=Operator message=Select Yes for a Left side weld, or select No for a Right Side weld. valueType=Boolean)
  sidewallchoice :=  (valueSource=Operator message=Is the sidewall 3/4 inch? valueType=Boolean)
  If sidewallchoice
    sidewall := 0.628
  Else 
    sidewall := 0.375
  MoveJ speed 60 deg/s, acceleration 80 deg/s^2 (useActiveTCP=true) feature=Base
    Waypoint Waypoint_46: TCP in base x=894.108 y=351.078 z=354.456 mm, rx=2.3264 ry=2.0525 rz=0.0574 rad; joints [-187.182, -67.294, 94.726, 57.522, -0.141, -88.018] deg
  Set NoAction tcp=pretend_w_top
  Script: Test_Teach_Position()
  Set NoAction tcp=pretend_w_top
  Script: kill threadId_Thread_1
  Script: Corner_Homing_45()
  Set NoAction tcp=pretend_welder
  SuppressedNode
    path1 := analyze_touchpoints(p11,p12,p21,p22,p3)
  SuppressedNode
    CallSubProgram
  SuppressedNode
    MoveJ speed 60 deg/s, acceleration 80 deg/s^2 (useActiveTCP=true) feature=Base
      Waypoint Waypoint_19: TCP in base x=-539.433 y=254.004 z=21.521 mm, rx=-1.7232 ry=0.9213 rz=1.7071 rad; joints [-41.97, -63.602, 146.502, 9.159, 84.533, 189.272] deg; TCP offset x=8.55 y=-271.52 z=102 mm, rx=1.2092 ry=-1.2092 rz=1.2092 rad
  If leftchoice≟ True
    pathturn := main_calculate_left_extended(p11,p12,p21,p22,p3,p13,p23,sidewall,tcp_pose_top)
    Script: extrude_knife3()
    Call move_path_3left
  Else 
    pathturn := main_calculate_right_extended(p11,p12,p21,p22,p3,p13,p23,sidewall,tcp_pose_top)
    Script: extrude_knife3()
    Script: move_path_3right()
  SuppressedNode
    Popup Message (haltProgram=false inputType=Variable) variable=pathturn
  MoveJ speed 60 deg/s, acceleration 80 deg/s^2 (useActiveTCP=true) feature=Base
    Waypoint Waypoint_46: TCP in base x=894.108 y=351.078 z=354.456 mm, rx=2.3264 ry=2.0525 rz=0.0574 rad; joints [-187.182, -67.294, 94.726, 57.522, -0.141, -88.018] deg; TCP offset x=-5.49 y=-328 z=106.39 mm, rx=1.2092 ry=-1.2092 rz=1.2092 rad
  SafeHome (positionOptionType=SPEED_AND_ACCELERATION speed=1.047198 acceleration=1.396263 nextMotionTime=2)
SubProgram move_path_3right (keepSynchronizedWithDisk=false) programFile=/programs/move_path_3right.urp
  'this is the path for Down, Over, then Back Around'
  ''
  SuppressedNode
    MoveJ speed 60 deg/s, acceleration 80 deg/s^2 (useActiveTCP=true) feature=Base
      Waypoint Waypoint_6: TCP in base x=-184.857 y=475.908 z=794.864 mm, rx=-0.225 ry=-1.9295 rz=0.6849 rad; joints [-137.383, -87.857, 120.236, 55.281, -50.736, -25.25] deg; TCP offset x=-5.053 y=-331.71 z=103.574 mm, rx=1.2092 ry=-1.2092 rz=1.2092 rad
      Waypoint Waypoint_1: TCP in base x=-161.037 y=970.524 z=722.042 mm, rx=-0.555 ry=0.1065 rz=0.3286 rad; joints [-74.895, -76.586, 126.53, 213.07, -169.134, 52.325] deg; TCP offset x=-4.211 y=-279.829 z=105.916 mm, rx=1.2092 ry=-1.2092 rz=1.2092 rad
      Waypoint Waypoint_7: TCP in base x=-689.651 y=138.963 z=230.691 mm, rx=-0.852 ry=-1.646 rz=1.646 rad; joints [-53.938, -86.03, 160.535, 285.425, -269.23, 90.049] deg
      SuppressedNode
        Waypoint Waypoint_1: TCP in base x=-1177.596 y=138.956 z=230.69 mm, rx=-0.852 ry=-1.646 rz=1.646 rad; joints [-20.637, -63.427, 120.718, 302.664, -235.94, 90.036] deg
      SuppressedNode
        Waypoint Waypoint_2: TCP in base x=-689.651 y=138.963 z=230.691 mm, rx=-0.852 ry=-1.646 rz=1.646 rad; joints [-53.938, -86.03, 160.535, 285.425, -269.23, 90.049] deg
      SuppressedNode
        Waypoint Waypoint_3: TCP in base x=-161.037 y=970.524 z=722.042 mm, rx=-0.555 ry=0.1065 rz=0.3286 rad; joints [-74.895, -76.586, 126.53, 213.07, -169.134, 52.325] deg
      SuppressedNode
        SafeHome (positionOptionType=SPEED_AND_ACCELERATION speed=1.047198 acceleration=1.396263 nextMotionTime=2)
  Script: align_ready_for_welding()
  ''
  p1 := pathturn[0]
  p2 := pathturn[1]
  p4 := pathturn[2]
  p5 := pathturn[3]
  pa1 := p[p1[0]+0.05,p1[1]+0.05,p1[2],p1[3],p1[4],p1[5]]
  MoveJ speed 20 deg/s, acceleration 80 deg/s^2 (useActiveTCP=true) feature=Base
    Waypoint Variable (Variable): variable=pa1
  MoveL speed 50 mm/s, acceleration 200 mm/s^2 (useActiveTCP=true) feature=Base
    Waypoint Variable (Variable): variable=p1
  Wait Sleep waitTime=8
  URCap WireTank Serial (WireTank Serial, WireTank, LLC) dataModel(NODE_TITLE=Serial Bridge uR1, Command=[252,82,49], QUERY=false, OUTPUT_ENTRY=Static, byte_array=true, Variable(key=OUTPUT_VARIABLE, variable=HwResp))
  URCap WireTank Serial (WireTank Serial, WireTank, LLC) dataModel(NODE_TITLE=Serial Bridge uR1, Command=[252,82,49], QUERY=false, byte_array=true, OUTPUT_ENTRY=Static, Variable(key=OUTPUT_VARIABLE, variable=HwResp))
  Wait Sleep waitTime=1
  SuppressedNode
    Script: turn_extrusion_on()
  Set DigitalOutput pin=digital_out[0]; digitalValue=1
  MoveL speed 10 mm/s, acceleration 100 mm/s^2 (useActiveTCP=true) feature=Base
    Waypoint Variable (Variable): variable=p2
  URCap WireTank Serial (WireTank Serial, WireTank, LLC) dataModel(QUERY=false, NODE_TITLE=Serial Bridge uR0, Command=[252,82,48], byte_array=true, OUTPUT_ENTRY=Static, Variable(key=OUTPUT_VARIABLE, variable=HwResp))
  Wait Sleep waitTime=0.5
  Set DigitalOutput pin=digital_out[0]; digitalValue=0
  MoveL speed 120 mm/s, acceleration 10 mm/s^2 (useActiveTCP=true) feature=Base
    Waypoint Variable (Variable): variable=p4
  URCap WireTank Serial (WireTank Serial, WireTank, LLC) dataModel(byte_array=true, NODE_TITLE=Serial Bridge uR1, Command=[252,82,49], QUERY=false, OUTPUT_ENTRY=Static, Variable(key=OUTPUT_VARIABLE, variable=HwResp))
  URCap WireTank Serial (WireTank Serial, WireTank, LLC) dataModel(NODE_TITLE=Serial Bridge uR1, Command=[252,82,49], QUERY=false, byte_array=true, OUTPUT_ENTRY=Static, Variable(key=OUTPUT_VARIABLE, variable=HwResp))
  Wait Sleep waitTime=1
  SuppressedNode
    Script: turn_extrusion_on()
  Set DigitalOutput pin=digital_out[0]; digitalValue=1
  MoveL speed 10 mm/s, acceleration 100 mm/s^2 (useActiveTCP=true) feature=Base
    Waypoint Variable (Variable): variable=p5
  URCap WireTank Serial (WireTank Serial, WireTank, LLC) dataModel(QUERY=false, NODE_TITLE=Serial Bridge uR0, Command=[252,82,48], OUTPUT_ENTRY=Static, byte_array=true, Variable(key=OUTPUT_VARIABLE, variable=HwResp))
  Wait Sleep waitTime=2
  Set DigitalOutput pin=digital_out[0]; digitalValue=0
  ''
  pret1 := p[p5[0]+.1,p5[1],p5[2],p5[3],p5[4],p5[5]]
  p_1 := pathturn[4]
  p_2 := pathturn[5]
  p_3 := pathturn[6]
  p_4 := pathturn[7]
  p_5 := pathturn[8]
  p_preheat := p[p_3[0]+.01,p_3[1],p_3[2],p_3[3],p_3[4],p_3[5]]
  p_pre_ret := p[p_1[0]+.03,p_1[1]+.03,p_1[2],p_1[3],p_1[4],p_1[5]]
  p_pre_ret2 := p[p_3[0]+.1,p_3[1],p_3[2],p_3[3],p_3[4],p_3[5]]
  'twist'
  MoveJ speed 80 deg/s, acceleration 80 deg/s^2 (useActiveTCP=true) feature=Base
    Waypoint Variable (Variable): variable=pret1
    Waypoint Waypoint_8: motionParameters(jointSpeed=1.047198 jointAcceleration=1.396263 cartesianSpeed=0.25 cartesianAcceleration=1.2); TCP in base x=-689.651 y=138.963 z=230.691 mm, rx=-0.852 ry=-1.646 rz=1.646 rad; joints [-53.938, -86.03, 160.535, 285.425, -269.23, 90.049] deg
    SuppressedNode
      Waypoint Waypoint_22: TCP in base x=-308.534 y=606.085 z=242.393 mm, rx=1.3699 ry=1.0669 rz=-1.2572 rad; joints [-84.142, -55.374, 92.791, 53.186, 94.965, 15.074] deg
  MoveJ speed 60 deg/s, acceleration 80 deg/s^2 (useActiveTCP=true) feature=Base
    Waypoint raa1: TCP in base x=-689.643 y=139.074 z=230.691 mm, rx=-0.8521 ry=-1.6459 rz=1.6459 rad; joints [-65.636, -88.39, 163.033, 285.277, -280.919, 90.061] deg; TCP offset x=-5.49 y=-328 z=106.39 mm, rx=1.2092 ry=-1.2092 rz=1.2092 rad
    Waypoint raa2: TCP in base x=-114.157 y=855.108 z=597.477 mm, rx=-0.5059 ry=0.3258 rz=0.3887 rad; joints [-71.965, -76.72, 138.376, 209.36, -156.862, 65.09] deg
    Waypoint raa3: TCP in base x=-308.547 y=387.798 z=242.407 mm, rx=1.9763 ry=0.3502 rz=-1.916 rad; joints [-108.471, -75.035, 126.793, 41.355, 93.912, 46.558] deg
    Waypoint raa4: TCP in base x=-733.576 y=77.691 z=242.41 mm, rx=1.9764 ry=0.3501 rz=-1.9161 rad; joints [-51.046, -76.954, 130.276, 41.633, 89.45, 103.864] deg
    SuppressedNode
      Waypoint Waypoint_2: TCP in base x=-308.546 y=606.076 z=242.404 mm, rx=1.3699 ry=1.0669 rz=-1.2572 rad; joints [-84.814, -53.028, 88.323, 55.251, 94.969, 14.398] deg
  'preheat'
  SuppressedNode
    MoveJ speed 60 deg/s, acceleration 80 deg/s^2 (useActiveTCP=true) feature=Base
      Waypoint Variable (Variable): variable=p_pre_ret
  MoveL speed 250 mm/s, acceleration 1200 mm/s^2 (useActiveTCP=true) feature=Base
    Waypoint Variable (Variable): variable=p_pre_ret2
    Waypoint Variable (Variable): variable=p_preheat
  Wait Sleep waitTime=6
  MoveL speed 250 mm/s, acceleration 1200 mm/s^2 (useActiveTCP=true) feature=Base
    Waypoint Variable (Variable): variable=p_pre_ret2
    Waypoint Variable (Variable): variable=p_pre_ret
  Set NoAction tcp=backofhole
  MoveL speed 50 mm/s, acceleration 1200 mm/s^2 (useActiveTCP=true) feature=Base
    Waypoint Variable (Variable): variable=p_1
  URCap WireTank Serial (WireTank Serial, WireTank, LLC) dataModel(NODE_TITLE=Serial Bridge uR1, Command=[252,82,49], QUERY=false, byte_array=true, OUTPUT_ENTRY=Static, Variable(key=OUTPUT_VARIABLE, variable=HwResp))
  URCap WireTank Serial (WireTank Serial, WireTank, LLC) dataModel(NODE_TITLE=Serial Bridge uR1, Command=[252,82,49], QUERY=false, byte_array=true, OUTPUT_ENTRY=Static, Variable(key=OUTPUT_VARIABLE, variable=HwResp))
  Wait Sleep waitTime=1
  Set DigitalOutput pin=digital_out[0]; digitalValue=1
  SuppressedNode
    Script: turn_extrusion_on()
  Wait Sleep waitTime=1
  MoveL speed 10 mm/s, acceleration 1200 mm/s^2 (useActiveTCP=true) feature=Base
    Waypoint Variable (Variable): variable=p_2
  MoveP speed 0.5 mm/s, acceleration 10 mm/s^2 (blendRadius=0.001 useActiveTCP=true) feature=Base
    CircleMove (OrientationMode=FIXED)
      Waypoint Variable (Variable): variable=p_3
      Waypoint Variable (Variable): variable=p_4
  MoveL speed 12 mm/s, acceleration 1200 mm/s^2 (useActiveTCP=true) feature=Base
    Waypoint Variable (Variable): variable=p_5
  URCap WireTank Serial (WireTank Serial, WireTank, LLC) dataModel(QUERY=false, NODE_TITLE=Serial Bridge uR0, Command=[252,82,48], OUTPUT_ENTRY=Static, byte_array=true, Variable(key=OUTPUT_VARIABLE, variable=HwResp))
  Wait Sleep waitTime=2
  Set DigitalOutput pin=digital_out[0]; digitalValue=0
  MoveL speed 250 mm/s, acceleration 1200 mm/s^2 (useActiveTCP=true) feature=Base
    Waypoint Waypoint_23: TCP in base x=-540.167 y=215.949 z=34.631 mm, rx=-1.5058 ry=1.0576 rz=1.5735 rad; joints [-26.452, -65.119, 143.749, 8.723, 85.674, 218.843] deg; TCP offset x=-4.211 y=-279.829 z=105.916 mm, rx=1.2092 ry=-1.2092 rz=1.2092 rad
  MoveJ speed 60 deg/s, acceleration 80 deg/s^2 (useActiveTCP=true) feature=Base
    Waypoint Waypoint_24: TCP in base x=-308.526 y=606.096 z=242.373 mm, rx=-2.1337 ry=0.3494 rz=2.1309 rad; joints [-107.196, -73.784, 125.643, 43.029, 90.975, 86.468] deg
    Waypoint Waypoint_39: TCP in base x=397.377 y=356.253 z=319.81 mm, rx=2.3163 ry=2.0576 rz=0.0741 rad; joints [-198.126, -117.851, 133.304, -13.01, -11.422, -6.036] deg; TCP offset x=-5.49 y=-328 z=106.39 mm, rx=1.2092 ry=-1.2092 rz=1.2092 rad
    'above waypoint is home'
SubProgram -> move_path_3left
SubProgram Test_Teach_Position (keepSynchronizedWithDisk=false) programFile=/programs/Test Teach Position.urp
  SuppressedNode
    MoveL speed 250 mm/s, acceleration 1200 mm/s^2 (useActiveTCP=true) feature=Base
      Waypoint Waypoint_1: TCP in base x=183.613 y=373.491 z=464.002 mm, rx=0 ry=3.1416 rz=0 rad; joints [-144.817, -120.486, 148.461, -117.931, -90.033, 125.101] deg; TCP offset x=0 y=0 z=19 mm, rx=0 ry=0 rz=0 rad
      'move welder up out of holder'
  MoveJ speed 60 deg/s, acceleration 80 deg/s^2 (useActiveTCP=false) tcp=TCP_1_plate; feature=Base
    Waypoint Waypoint_40: TCP in base x=360.688 y=270.12 z=646.145 mm, rx=0.0578 ry=2.126 rz=2.1341 rad; joints [-198.126, -117.852, 133.303, -13.01, -11.422, -6.036] deg
    'above waypoint is home'
    Waypoint Waypoint_2: TCP in base x=-548.957 y=386.285 z=143.71 mm, rx=1.5708 ry=0 rz=0 rad; joints [-60.253, -57.926, 123.544, -65.529, -60.311, -0.099] deg
  freedrive_m_var := False
  freedrive_m_var := True
  Popup Message (haltProgram=false message=Move the TCP to the top of the weld, then click 'Continue' inputType=Text)
  tcp_pose_top := get_actual_tcp_pose()
  Popup Message (haltProgram=false message=Move the TCP to the corner of the tank, then click 'Continue' inputType=Text)
  tcp_pose := get_actual_tcp_pose()
  freedrive_m_var := False
  Wait Sleep waitTime=0.25
  Script: sync()
SubProgram align_tcp_left (keepSynchronizedWithDisk=false) programFile=/programs/align_tcp_left.urp
  'this program aligns the tcp parallel to the y direction'
  cp := get_actual_tcp_pose()
  aligned_y_pose := p[cp[0],cp[1],cp[2],1.570796,0,0]
  MoveJ speed 60 deg/s, acceleration 80 deg/s^2 (useActiveTCP=true) feature=Base
    Waypoint Variable (Variable): variable=aligned_y_pose
SubProgram extrude_knife3 (keepSynchronizedWithDisk=false) programFile=/programs/extrude_knife3.urp
  SuppressedNode
    SafeHome (positionOptionType=SPEED_AND_ACCELERATION speed=1.047198 acceleration=1.396263 nextMotionTime=2)
  Set NoAction tcp=pretend_welder
  MoveJ speed 60 deg/s, acceleration 80 deg/s^2 (useActiveTCP=true) feature=Base
    Waypoint Waypoint_20: TCP in base x=397.38 y=356.254 z=319.821 mm, rx=2.3163 ry=2.0576 rz=0.0741 rad; joints [-198.126, -117.851, 133.303, -13.009, -11.422, -6.035] deg; TCP offset x=-5.49 y=-328 z=106.39 mm, rx=1.2092 ry=-1.2092 rz=1.2092 rad
    'above waypoint is home'
  'move above bucket'
  MoveJ speed 60 deg/s, acceleration 80 deg/s^2 (useActiveTCP=true) feature=Base
    Waypoint Waypoint_3: TCP in base x=454.852 y=405.449 z=64.015 mm, rx=2.3168 ry=2.0514 rz=0.0767 rad; joints [-187.624, -89.406, 141.395, -19.732, -0.818, -36.116] deg
  'extrude out a foot'
  SuppressedNode
    URCap WireTank Serial (WireTank Serial, WireTank, LLC) dataModel(byte_array=true, NODE_TITLE=Serial Bridge uR1, Command=[252,82,49], QUERY=false, OUTPUT_ENTRY=Static, Variable(key=OUTPUT_VARIABLE, variable=HwResp))
  Script: turn_extrusion_on()
  URCap WireTank Serial (WireTank Serial, WireTank, LLC) dataModel(NODE_TITLE=Serial Bridge uR1, Command=[252,82,49], QUERY=false, OUTPUT_ENTRY=Static, byte_array=true, Variable(key=OUTPUT_VARIABLE, variable=HwResp))
  Set DigitalOutput pin=digital_out[0]; digitalValue=1
  Wait Sleep waitTime=24
  URCap WireTank Serial (WireTank Serial, WireTank, LLC) dataModel(QUERY=false, NODE_TITLE=Serial Bridge uR0, Command=[252,82,48], byte_array=true, OUTPUT_ENTRY=Static, Variable(key=OUTPUT_VARIABLE, variable=HwResp))
  Wait Sleep waitTime=1
  Set DigitalOutput pin=digital_out[0]; digitalValue=0
  'slice'
  MoveL speed 30 mm/s, acceleration 50 mm/s^2 (useActiveTCP=true) feature=Base
    Waypoint Waypoint_21: TCP in base x=439.065 y=405.452 z=65.996 mm, rx=2.3168 ry=2.0514 rz=0.0766 rad; joints [-187.962, -93.321, 143.386, -27.168, -1.131, -26.752] deg
    Waypoint Waypoint_42: TCP in base x=419.01 y=404.851 z=65.995 mm, rx=2.3096 ry=2.0447 rz=0.0891 rad; joints [-188.553, -97.485, 146.002, -33.769, -1.69, -19.324] deg
    Waypoint Waypoint_43: TCP in base x=417.012 y=405.435 z=65.003 mm, rx=2.3169 ry=2.0513 rz=0.0766 rad; joints [-188.493, -97.025, 145.794, -33.21, -1.638, -19.415] deg
    Waypoint Waypoint_44: TCP in base x=413.072 y=405.431 z=68 mm, rx=2.3168 ry=2.0513 rz=0.0767 rad; joints [-188.596, -97.887, 146.02, -33.517, -1.738, -18.475] deg
    Waypoint Waypoint_74: TCP in base x=389.999 y=405.444 z=68.005 mm, rx=2.3169 ry=2.0514 rz=0.0766 rad; joints [-189.248, -101.07, 148.002, -36.337, -2.38, -14.447] deg
  MoveJ speed 60 deg/s, acceleration 80 deg/s^2 (useActiveTCP=true) feature=Base
    Waypoint Waypoint_45: TCP in base x=397.38 y=356.254 z=319.821 mm, rx=2.3163 ry=2.0576 rz=0.0741 rad; joints [-198.126, -117.851, 133.303, -13.009, -11.422, -6.035] deg
    'above waypoint is home'
  SuppressedNode
    SafeHome (positionOptionType=SPEED_AND_ACCELERATION speed=1.047198 acceleration=1.396263 nextMotionTime=2)
SubProgram align_tcp_forward (keepSynchronizedWithDisk=false) programFile=/programs/align_tcp_forward.urp
  'this program aligns the tcp parallel to the y direction'
  cp := get_actual_tcp_pose()
  aligned_y_pose := p[cp[0],cp[1],cp[2],0,-1.570796,0]
  MoveJ speed 60 deg/s, acceleration 80 deg/s^2 (useActiveTCP=true) feature=Base
    Waypoint Variable (Variable): variable=aligned_y_pose
SubProgram align_tcp_up (keepSynchronizedWithDisk=false) programFile=/programs/align_tcp_up.urp
  'this program aligns the tcp parallel to the y direction'
  cp := get_actual_tcp_pose()
  aligned_y_pose := p[cp[0],cp[1],cp[2],0,0,0]
  MoveJ speed 60 deg/s, acceleration 80 deg/s^2 (useActiveTCP=true) feature=Base
    Waypoint Variable (Variable): variable=aligned_y_pose
SubProgram align_ready_for_welding (keepSynchronizedWithDisk=false) programFile=/programs/align_ready_for_welding.urp
  'this program takes the welder from home to a position alined ready for welding (vertically down)'
  MoveJ speed 60 deg/s, acceleration 80 deg/s^2 (useActiveTCP=true) feature=Base
    Waypoint oldhome: TCP in base x=397.684 y=356.251 z=315.247 mm, rx=2.3163 ry=2.0576 rz=0.0741 rad; joints [-198.127, -117.852, 133.304, -13.011, -11.422, -6.036] deg; TCP offset x=-5.492 y=-332.581 z=106.393 mm, rx=1.2092 ry=-1.2092 rz=1.2092 rad
    Waypoint Waypoint_34: TCP in base x=695.155 y=367.452 z=502.522 mm, rx=2.0931 ry=1.8575 rz=0.3088 rad; joints [-186.178, -111.085, 133.076, 228.143, -3.264, 87.587] deg
    Waypoint Waypoint_35: TCP in base x=687.528 y=415.166 z=537.921 mm, rx=2.1271 ry=1.9299 rz=0.4701 rad; joints [-186.178, -111.085, 133.077, 228.144, -355.12, 87.586] deg
    Waypoint Waypoint_36: TCP in base x=-693.756 y=141.369 z=218.585 mm, rx=-0.852 ry=-1.646 rz=1.646 rad; joints [-66.082, -85.509, 163.4, 282.028, -281.373, 90.065] deg
SubProgram Corner_Homing_45 (keepSynchronizedWithDisk=false) programFile=/programs/Corner Homing 45.urp
  'Use this program when tool is already positioned close to corner at 45deg'
  'tool flange will seek all 3 sides. will save those 5 locs in p__'
  Set NoAction tcp=pretend_w_top
  'dummy move below for debug'
  SuppressedNode
    SafeHome (positionOptionType=SPEED_AND_ACCELERATION speed=1.047198 acceleration=1.396263 nextMotionTime=2)
  SuppressedNode
    MoveJ speed 60 deg/s, acceleration 80 deg/s^2 (useActiveTCP=true) feature=Base
      Waypoint Waypoint_1: TCP in base x=-726.76 y=313.857 z=-3.219 mm, rx=-0.1302 ry=-1.6605 rz=-0.1403 rad; joints [-65.067, -50.619, 153.092, -93.35, 35.027, 81.724] deg; TCP offset x=0 y=0 z=246 mm, rx=0 ry=0 rz=0 rad
      Waypoint Waypoint_2: TCP in base x=-1013.668 y=283.774 z=13.404 mm, rx=-0.1302 ry=-1.6605 rz=-0.1403 rad; joints [-36.803, -53.188, 133.142, -74.065, 63.057, 86.565] deg
  Wait Sleep waitTime=1
  tp := get_actual_tcp_pose()
  SuppressedNode
    Script file /programs/analyze_touchpoints.script
      | # this file creates the function for analyzing touchpoints
      | # define pi
      | pi = 3.1415926535
      | 
      | # this is the main entry point for calculations.
      | # it takes in the 5 points, analyzes the shape of the box, and then calculates path points and returns them
      | # specifically for Down, Over, then Around (DOtA)
      | # specifically for right-sided boxes (vertical weld on right side of edge)
      | def main_calculate_right(p11, p12, p21, p22, p3, p13, p23, chamferover):
      |     struct1 = analyze_touchpoints_only(p11, p12, p21, p22, p3)
      |     list1 = analyze_vertical_touchpoints(p11, p12, p13, p21, p22, p23, p3)
      |     struct2 = calculate_DOtA_points_right(struct1, list1, chamferover)
      |     validity = check_validity_right(struct1, struct2)
      |     return struct2
      | end
      | 
      | # this is the main entry point for calculations.
      | # it takes in the 5 points, analyzes the shape of the box, and then calculates path points and returns them
      | # specifically for Down, Over, then Around (DOtA)
      | # specifically for left-sided boxes (vertical weld on left side of edge)
      | def main_calculate_left(p11, p12, p21, p22, p3, p13, p23, chamferover):
      |     struct1 = analyze_touchpoints_only(p11, p12, p21, p22, p3)
      |     list1 = analyze_vertical_touchpoints(p11, p12, p13, p21, p22, p23, p3)
      |     struct2 = calculate_DOtA_points_left(struct1, list1, chamferover)
      |     validity = check_validity_left(struct1, struct2)
      |     return struct2
      | end
      | 
      | # this is the main entry point for calculations, for Floor Corner Extended.
      | # it takes in the 7 touchpoints, analyzes the shape of the box.
      | # takes in the user defined point for the top of the weld (tcp_pose_top) and then calculates path points
      | # loopingly tries to calculate the extension along the sidewall that fulfills get_inverse_kin_has_solution() and provides the farthest extension possible
      | # returns the pathpoints
      | # specifically for Down, Over, then Around (DOtA)
      | # specifically for right-sided boxes (vertical weld on right side of edge)
      | def main_calculate_right_extended(p11, p12, p21, p22, p3, p13, p23, chamferover, tcp_pose_top):
      |     struct1 = analyze_touchpoints_only(p11, p12, p21, p22, p3)
      |     list1 = analyze_vertical_touchpoints(p11, p12, p13, p21, p22, p23, p3)
      |     struct2 = calculate_DOtA_points_right_extended(struct1, list1, chamferover, tcp_pose_top)
      |     validity = check_validity_right(struct1, struct2)
      |     return struct2
      | end
      | 
      | # this is the main entry point for calculations, for Floor Corner Extended.
      | # it takes in the 7 touchpoints, analyzes the shape of the box.
      | # takes in the user defined point for the top of the weld (tcp_pose_top) and then calculates path points
      | # loopingly tries to calculate the extension along the sidewall that fulfills get_inverse_kin_has_solution() and provides the farthest extension possible
      | # returns the pathpoints
      | # specifically for Down, Over, then Around (DOtA)
      | # specifically for left-sided boxes (vertical weld on left side of edge)
      | def main_calculate_left_extended(p11, p12, p21, p22, p3, p13, p23, chamferover, tcp_pose_top):
      |     struct1 = analyze_touchpoints_only(p11, p12, p21, p22, p3)
      |     list1 = analyze_vertical_touchpoints(p11, p12, p13, p21, p22, p23, p3)
      |     struct2 = calculate_DOtA_points_left_extended(struct1, list1, chamferover, tcp_pose_top)
      |     validity = check_validity_left(struct1, struct2)
      |     return struct2
      | end
      | 
      | # it takes 5 arguments as points
      | # it returns a struct containing: (pointintersect, pointapproach1, pointapproach2, point1, point2, point3, point4, point5, pointreturn1, heading1, heading2, heading3, path2r1, path2r2, path2l1, path2l2)
      | # specifically for Around then Up (AtU)
      | def analyze_touchpoints(p11, p12, p21, p22, p3):
      |   # FIND THE INTERSECTION
      |   # comment get the z
      |   zcoord=p3[2]
      | 
      |   # get the raw points from the first line
      |   l1p1x=p11[0]
      |   l1p1y=p11[1]
      |   l1p2x=p12[0]
      |   l1p2y=p12[1]
      | 
      |   # equate the first line in 2d space
      |   ml1 = (l1p2y-l1p1y) / (l1p2x-l1p1x)
      | 
      |   # b = y - mx
      |   bl1 = l1p1y - ml1 * l1p1x
      | 
      |   # get the raw points from the second line
      |   l2p1x=p21[0]
      |   l2p1y=p21[1]
      |   l2p2x=p22[0]
      |   l2p2y=p22[1]
      | 
      |   # equate the second line in 2d space
      |   ml2 = (l2p2y-l2p1y) / (l2p2x-l2p1x)
      | 
      |   # b = y - mx
      |   bl2 = l2p1y - ml2 * l2p1x
      | 
      | 
      |   # find the intersection of the two lines
      |   # m1x+b1 = m2x+b2
      |   # m1x - m2x = b2 - b1
      |   # x = (b2-b1) / (m1-m2)
      |   xintersect = (bl2-bl1) / (ml1-ml2)
      |   yintersect = ml1 * xintersect + bl1
      | 
      |   #FIND THE VECTORS
      |   #define a vector from the intersection to the second point on the first line
      |   l1delxfull = l1p2x - xintersect
      |   l1delyfull = l1p2y - yintersect
      | 
      |   l1delmag = sqrt(l1delxfull*l1delxfull + l1delyfull*l1delyfull)
      | 
      |   l1delxunit = l1delxfull / l1delmag
      |   l1delyunit = l1delyfull / l1delmag
      | 
      |   #define a vector from the intersection to the second point on the second line
      |   l2delxfull = l2p2x - xintersect
      |   l2delyfull = l2p2y - yintersect
      | 
      |   l2delmag = sqrt(l2delxfull*l2delxfull + l2delyfull*l2delyfull)
      | 
      |   l2delxunit = l2delxfull / l2delmag
      |   l2delyunit = l2delyfull / l2delmag
      | 
      |   # FIND THE FOUR POINTS ON THE LINES
      |   # find locations 8 inches away from  intersect point
      |   # CONST
      |   welddistance = 8
      |   roundoverdistance = 0.05
      |   zup = .375
      |   # inches
      |   wd = welddistance * 25.4 / 1000
      |   rod = roundoverdistance * 25.4 / 1000
      |   zup = zup * 25.4 / 1000
      | 
      |   # now we have the unit vector. extend the weld distance from the intersection
      |   x = xintersect + l1delxunit * wd
      |   y = yintersect + l1delyunit * wd
      |   z = zcoord + zup
      | 
      |   point1 = p[x,y,z,1.570796,0,0] # dummy orientation for now
      | 
      |   x = xintersect + l1delxunit * rod
      |   y = yintersect + l1delyunit * rod
      | 
      |   point2 = p[x,y,z,1.570796,0,0]
      | 
      |   # now we have the unit vector. extend the weld distance from the intersection
      |   x = xintersect + l2delxunit * wd
      |   y = yintersect + l2delyunit * wd
      | 
      |   point5 = p[x,y,z,0,-1.570796,0]
      | 
      |   x = xintersect + l2delxunit * rod
      |   y = yintersect + l2delyunit * rod
      | 
      |   point4 = p[x,y,z,0,-1.570796,0]
      | 
      |   #DEFINE APPROACH POINTS
      |   pointintersect = p[xintersect,yintersect,zcoord,0,0,0]
      |   pointapproach1 = p[xintersect+0.1,yintersect+0.1,z,1.570796,0,0]
      |   pointapproach2 = p[point1[0], point1[1]+0.1, point1[2], point1[3], point1[4], point1[5]]
      |   pointreturn1 = p[point5[0]+0.1, point5[1], point5[2], point5[3], point5[4], point5[5]]
      | 
      |   #FIND HEADINGS
      |   #for each heading, find the angle of the line with respect to the pos x axis. then add/subtract 90 degrees because you want to be perpendicular to that
      |   headingvector1 = convert_uv_to_heading(l1delxunit, l1delyunit)
      |   headingvector2 = convert_uv_to_heading(l2delxunit, l2delyunit)
      |   # find halfway heading
